LIN {X 0.107,Y -668.681,Z 738.565,A 0.000,B 0.000,C 90.000,E1 317.676} C_DIS
LIN {X 0.186,Y -672.664,Z 738.558,A 0.000,B 0.000,C 90.000,E1 316.458} C_DIS
LIN {X 0.302,Y -676.399,Z 738.552,A 0.000,B 0.000,C 90.000,E1 315.243} C_DIS
LIN {X -0.045,Y -679.125,Z 738.546,A 0.000,B 0.000,C 90.000,E1 314.312} C_DIS
LIN {X 0.190,Y -682.249,Z 738.540,A 0.000,B 0.000,C 90.000,E1 313.095} C_DIS
LIN {X 0.341,Y -684.050,Z 738.536,A 0.000,B 0.000,C 90.000,E1 312.366} C_DIS
LIN {X -0.296,Y -686.830,Z 738.529,A 0.000,B 0.000,C 90.000,E1 311.229} C_DIS
LIN {X 0.079,Y -689.190,Z 738.522,A 0.000,B 0.000,C 90.000,E1 310.011} C_DIS
LIN {X -0.016,Y -690.783,Z 738.517,A 0.000,B 0.000,C 90.000,E1 309.072} C_DIS
LIN {X 0.345,Y -692.184,Z 738.512,A 0.000,B 0.000,C 90.000,E1 308.096} C_DIS
LIN {X 0.292,Y -693.400,Z 738.507,A 0.000,B 0.000,C 90.000,E1 307.156} C_DIS
LIN {X -0.101,Y -694.755,Z 738.500,A 0.000,B 0.000,C 90.000,E1 306.011} C_DIS
LIN {X 0.435,Y -695.668,Z 738.495,A 0.000,B 0.000,C 90.000,E1 305.025} C_DIS
LIN {X -0.332,Y -696.670,Z 738.488,A 0.000,B 0.000,C 90.000,E1 303.913} C_DIS
LIN {X 0.362,Y -697.989,Z 738.479,A 0.000,B 0.000,C 90.000,E1 302.212} C_DIS
LIN {X 0.208,Y -698.942,Z 738.473,A 0.000,B 0.000,C 90.000,E1 301.052} C_DIS
LIN {X 0.041,Y -699.423,Z 738.467,A 0.000,B 0.000,C 90.000,E1 300.129} C_DIS
LIN {X 0.151,Y -699.766,Z 738.461,A 0.000,B 0.000,C 90.000,E1 298.949} C_DIS
LIN {X 0.265,Y -700.096,Z 738.454,A 0.000,B 0.000,C 90.000,E1 297.769} C_DIS
LIN {X 0.057,Y -700.510,Z 738.448,A 0.000,B 0.000,C 90.000,E1 296.616} C_DIS
LIN {X 0.130,Y -701.206,Z 738.440,A 0.000,B 0.000,C 90.000,E1 295.207} C_DIS
LIN {X -0.253,Y -701.147,Z 738.438,A 0.000,B 0.000,C 90.000,E1 294.771} C_DIS
LIN {X 0.020,Y -700.966,Z 738.436,A 0.000,B 0.000,C 90.000,E1 294.515} C_DIS
LIN {X -0.362,Y -700.003,Z 738.434,A 0.000,B 0.000,C 90.000,E1 294.079} C_DIS
LIN {X -0.093,Y -699.108,Z 738.432,A 0.000,B 0.000,C 90.000,E1 293.823} C_DIS
LIN {X -0.107,Y -697.250,Z 738.431,A 0.000,B 0.000,C 90.000,E1 293.590} C_DIS
LIN {X 0.281,Y -694.168,Z 738.429,A 0.000,B 0.000,C 90.000,E1 293.206} C_DIS
LIN {X -0.231,Y -692.628,Z 738.428,A 0.000,B 0.000,C 90.000,E1 293.131} C_DIS
LIN {X -0.206,Y -690.549,Z 738.428,A 0.000,B 0.000,C 90.000,E1 293.025} C_DIS
LIN {X 0.164,Y -686.427,Z 738.427,A 0.000,B 0.000,C 90.000,E1 292.823} C_DIS
LIN {X 0.124,Y -682.661,Z 738.426,A 0.000,B 0.000,C 90.000,E1 292.695} C_DIS
LIN {X -0.149,Y -676.703,Z 738.425,A 0.000,B 0.000,C 90.000,E1 292.567} C_DIS
LIN {X -0.265,Y -668.924,Z 738.425,A 0.000,B 0.000,C 90.000,E1 292.461} C_DIS
LIN {X -0.069,Y -659.282,Z 738.424,A 0.000,B 0.000,C 90.000,E1 292.333} C_DIS
LIN {X -0.387,Y -645.945,Z 738.423,A 0.000,B 0.000,C 90.000,E1 292.153} C_DIS
LIN {X 0.142,Y -632.515,Z 738.421,A 0.000,B 0.000,C 90.000,E1 291.844} C_DIS
LIN {X 0.064,Y -619.307,Z 738.420,A 0.000,B 0.000,C 90.000,E1 291.535} C_DIS
LIN {X 0.213,Y -588.192,Z 738.415,A 0.000,B 0.000,C 90.000,E1 290.663} C_DIS
LIN {X -0.258,Y -574.047,Z 738.413,A 0.000,B 0.000,C 90.000,E1 290.301} C_DIS
LIN {X 0.173,Y -566.696,Z 738.412,A 0.000,B 0.000,C 90.000,E1 290.066} C_DIS
LIN {X 0.081,Y -561.198,Z 738.411,A 0.000,B 0.000,C 90.000,E1 289.885} C_DIS
LIN {X 0.104,Y -556.813,Z 738.409,A 0.000,B 0.000,C 90.000,E1 289.631} C_DIS
LIN {X 0.047,Y -556.755,Z 738.409,A 0.000,B 0.000,C 90.000,E1 289.631} C_DIS
LIN {X 0.005,Y -555.577,Z 738.408,A 0.000,B 0.000,C 90.000,E1 289.450} C_DIS
LIN {X -0.006,Y -554.906,Z 738.406,A 0.000,B 0.000,C 90.000,E1 289.033} C_DIS
LIN {X 0.300,Y -554.456,Z 738.398,A 0.000,B 0.000,C 90.000,E1 287.692} C_DIS
LIN {X 0.241,Y -553.803,Z 738.389,A 0.000,B 0.000,C 90.000,E1 286.024} C_DIS
LIN {X -0.248,Y -553.121,Z 738.378,A 0.000,B 0.000,C 90.000,E1 284.120} C_DIS
LIN {X 0.178,Y -552.515,Z 738.367,A 0.000,B 0.000,C 90.000,E1 282.119} C_DIS
LIN {X 0.126,Y -552.034,Z 738.360,A 0.000,B 0.000,C 90.000,E1 280.725} C_DIS
LIN {X 0.171,Y -551.422,Z 738.352,A 0.000,B 0.000,C 90.000,E1 279.321} C_DIS
LIN {X 0.240,Y -550.474,Z 738.341,A 0.000,B 0.000,C 90.000,E1 277.352} C_DIS
LIN {X 0.211,Y -549.573,Z 738.330,A 0.000,B 0.000,C 90.000,E1 275.391} C_DIS
LIN {X -0.028,Y -548.987,Z 738.322,A 0.000,B 0.000,C 90.000,E1 274.012} C_DIS
LIN {X -0.214,Y -547.965,Z 738.311,A 0.000,B 0.000,C 90.000,E1 272.064} C_DIS
LIN {X -0.008,Y -547.441,Z 738.305,A 0.000,B 0.000,C 90.000,E1 270.917} C_DIS
LIN {X 0.221,Y -546.611,Z 738.297,A 0.000,B 0.000,C 90.000,E1 269.484} C_DIS
LIN {X -0.058,Y -545.522,Z 738.288,A 0.000,B 0.000,C 90.000,E1 267.822} C_DIS
LIN {X 0.248,Y -544.272,Z 738.277,A 0.000,B 0.000,C 90.000,E1 265.812} C_DIS
LIN {X -0.075,Y -543.297,Z 738.269,A 0.000,B 0.000,C 90.000,E1 264.432} C_DIS
LIN {X 0.189,Y -542.025,Z 738.260,A 0.000,B 0.000,C 90.000,E1 262.704} C_DIS
LIN {X -0.126,Y -540.901,Z 738.252,A 0.000,B 0.000,C 90.000,E1 261.319} C_DIS
LIN {X 0.219,Y -539.453,Z 738.242,A 0.000,B 0.000,C 90.000,E1 259.577} C_DIS
LIN {X 0.167,Y -537.839,Z 738.231,A 0.000,B 0.000,C 90.000,E1 257.589} C_DIS
LIN {X 0.076,Y -536.590,Z 738.223,A 0.000,B 0.000,C 90.000,E1 256.172} C_DIS
LIN {X -0.086,Y -535.398,Z 738.217,A 0.000,B 0.000,C 90.000,E1 255.046} C_DIS
LIN {X -0.074,Y -533.864,Z 738.209,A 0.000,B 0.000,C 90.000,E1 253.614} C_DIS
LIN {X -0.092,Y -532.365,Z 738.201,A 0.000,B 0.000,C 90.000,E1 252.181} C_DIS
LIN {X -0.168,Y -531.064,Z 738.195,A 0.000,B 0.000,C 90.000,E1 251.040} C_DIS
LIN {X -0.093,Y -529.518,Z 738.188,A 0.000,B 0.000,C 90.000,E1 249.880} C_DIS
LIN {X 0.141,Y -527.596,Z 738.180,A 0.000,B 0.000,C 90.000,E1 248.411} C_DIS
LIN {X 0.185,Y -526.349,Z 738.175,A 0.000,B 0.000,C 90.000,E1 247.539} C_DIS
LIN {X 0.236,Y -523.743,Z 738.166,A 0.000,B 0.000,C 90.000,E1 245.793} C_DIS
LIN {X -0.029,Y -520.893,Z 738.156,A 0.000,B 0.000,C 90.000,E1 244.076} C_DIS
LIN {X -0.160,Y -518.891,Z 738.150,A 0.000,B 0.000,C 90.000,E1 242.922} C_DIS
LIN {X 0.131,Y -516.673,Z 738.143,A 0.000,B 0.000,C 90.000,E1 241.719} C_DIS
LIN {X 0.080,Y -513.766,Z 738.135,A 0.000,B 0.000,C 90.000,E1 240.255} C_DIS
LIN {X -0.017,Y -510.889,Z 738.127,A 0.000,B 0.000,C 90.000,E1 238.791} C_DIS
LIN {X 0.201,Y -508.495,Z 738.120,A 0.000,B 0.000,C 90.000,E1 237.582} C_DIS
LIN {X -0.049,Y -505.942,Z 738.113,A 0.000,B 0.000,C 90.000,E1 236.421} C_DIS
LIN {X 0.251,Y -502.660,Z 738.105,A 0.000,B 0.000,C 90.000,E1 234.895} C_DIS
LIN {X 0.074,Y -499.029,Z 738.097,A 0.000,B 0.000,C 90.000,E1 233.417} C_DIS
LIN {X 0.126,Y -495.165,Z 738.089,A 0.000,B 0.000,C 90.000,E1 231.904} C_DIS
LIN {X -0.284,Y -491.468,Z 738.080,A 0.000,B 0.000,C 90.000,E1 230.436} C_DIS
LIN {X 0.245,Y -487.936,Z 738.072,A 0.000,B 0.000,C 90.000,E1 228.852} C_DIS
LIN {X -0.125,Y -481.804,Z 738.056,A 0.000,B 0.000,C 90.000,E1 226.134} C_DIS
LIN {X 0.073,Y -477.123,Z 738.044,A 0.000,B 0.000,C 90.000,E1 223.947} C_DIS
LIN {X -0.037,Y -473.885,Z 738.036,A 0.000,B 0.000,C 90.000,E1 222.405} C_DIS
LIN {X 0.107,Y -470.495,Z 738.027,A 0.000,B 0.000,C 90.000,E1 220.825} C_DIS
LIN {X 0.156,Y -464.903,Z 738.013,A 0.000,B 0.000,C 90.000,E1 218.302} C_DIS
LIN {X 0.091,Y -460.160,Z 738.001,A 0.000,B 0.000,C 90.000,E1 216.091} C_DIS
LIN {X -0.258,Y -455.010,Z 737.986,A 0.000,B 0.000,C 90.000,E1 213.579} C_DIS
LIN {X 0.008,Y -452.628,Z 737.979,A 0.000,B 0.000,C 90.000,E1 212.260} C_DIS
LIN {X -0.078,Y -448.964,Z 737.969,A 0.000,B 0.000,C 90.000,E1 210.335} C_DIS
LIN {X 0.144,Y -445.421,Z 737.958,A 0.000,B 0.000,C 90.000,E1 208.359} C_DIS
LIN {X -0.034,Y -442.971,Z 737.950,A 0.000,B 0.000,C 90.000,E1 207.078} C_DIS
LIN {X -0.209,Y -439.876,Z 737.941,A 0.000,B 0.000,C 90.000,E1 205.463} C_DIS
LIN {X -0.005,Y -436.307,Z 737.930,A 0.000,B 0.000,C 90.000,E1 203.462} C_DIS
LIN {X 0.123,Y -433.167,Z 737.921,A 0.000,B 0.000,C 90.000,E1 201.791} C_DIS
LIN {X 0.207,Y -428.839,Z 737.908,A 0.000,B 0.000,C 90.000,E1 199.450} C_DIS
LIN {X 0.082,Y -425.100,Z 737.897,A 0.000,B 0.000,C 90.000,E1 197.457} C_DIS
LIN {X -0.095,Y -422.490,Z 737.890,A 0.000,B 0.000,C 90.000,E1 196.134} C_DIS
LIN {X 0.004,Y -417.440,Z 737.875,A 0.000,B 0.000,C 90.000,E1 193.411} C_DIS
LIN {X -0.006,Y -413.905,Z 737.863,A 0.000,B 0.000,C 90.000,E1 191.366} C_DIS
LIN {X -0.044,Y -409.097,Z 737.848,A 0.000,B 0.000,C 90.000,E1 188.624} C_DIS
LIN {X -0.001,Y -406.349,Z 737.838,A 0.000,B 0.000,C 90.000,E1 186.891} C_DIS
LIN {X -0.200,Y -401.138,Z 737.819,A 0.000,B 0.000,C 90.000,E1 183.440} C_DIS
LIN {X 0.191,Y -397.074,Z 737.801,A 0.000,B 0.000,C 90.000,E1 180.229} C_DIS
LIN {X 0.167,Y -394.437,Z 737.788,A 0.000,B 0.000,C 90.000,E1 177.764} C_DIS
LIN {X 0.080,Y -391.977,Z 737.774,A 0.000,B 0.000,C 90.000,E1 175.298} C_DIS
LIN {X -0.138,Y -389.590,Z 737.756,A 0.000,B 0.000,C 90.000,E1 172.129} C_DIS
LIN {X 0.182,Y -388.175,Z 737.738,A 0.000,B 0.000,C 90.000,E1 168.870} C_DIS
LIN {X -0.080,Y -387.020,Z 737.722,A 0.000,B 0.000,C 90.000,E1 166.047} C_DIS
LIN {X 0.160,Y -386.296,Z 737.709,A 0.000,B 0.000,C 90.000,E1 163.504} C_DIS
LIN {X -0.177,Y -385.941,Z 737.697,A 0.000,B 0.000,C 90.000,E1 161.402} C_DIS
LIN {X 0.070,Y -385.662,Z 737.687,A 0.000,B 0.000,C 90.000,E1 159.571} C_DIS
LIN {X 0.113,Y -385.332,Z 737.675,A 0.000,B 0.000,C 90.000,E1 157.411} C_DIS
LIN {X -0.061,Y -385.252,Z 737.657,A 0.000,B 0.000,C 90.000,E1 154.204} C_DIS
LIN {X -0.062,Y -386.656,Z 737.631,A 0.000,B 0.000,C 90.000,E1 149.537} C_DIS
LIN {X -0.080,Y -389.021,Z 737.611,A 0.000,B 0.000,C 90.000,E1 145.960} C_DIS
LIN {X -0.062,Y -393.045,Z 737.591,A 0.000,B 0.000,C 90.000,E1 142.396} C_DIS
LIN {X 0.038,Y -395.333,Z 737.583,A 0.000,B 0.000,C 90.000,E1 140.964} C_DIS
LIN {X 0.017,Y -397.610,Z 737.577,A 0.000,B 0.000,C 90.000,E1 139.908} C_DIS
LIN {X -0.083,Y -399.603,Z 737.573,A 0.000,B 0.000,C 90.000,E1 139.218} C_DIS
LIN {X 0.085,Y -401.742,Z 737.570,A 0.000,B 0.000,C 90.000,E1 138.609} C_DIS
LIN {X 0.026,Y -405.333,Z 737.566,A 0.000,B 0.000,C 90.000,E1 137.919} C_DIS
LIN {X 0.203,Y -408.142,Z 737.564,A 0.000,B 0.000,C 90.000,E1 137.472} C_DIS
LIN {X -0.041,Y -413.068,Z 737.561,A 0.000,B 0.000,C 90.000,E1 136.905} C_DIS
LIN {X -0.026,Y -430.952,Z 737.550,A 0.000,B 0.000,C 90.000,E1 135.081} C_DIS
LIN {X -0.178,Y -447.096,Z 737.542,A 0.000,B 0.000,C 90.000,E1 133.542} C_DIS
LIN {X 0.034,Y -454.423,Z 737.538,A 0.000,B 0.000,C 90.000,E1 132.813} C_DIS
LIN {X 0.015,Y -465.875,Z 737.532,A 0.000,B 0.000,C 90.000,E1 131.676} C_DIS
LIN {X -0.272,Y -475.659,Z 737.526,A 0.000,B 0.000,C 90.000,E1 130.701} C_DIS
LIN {X 0.068,Y -482.496,Z 737.522,A 0.000,B 0.000,C 90.000,E1 129.930} C_DIS
LIN {X -0.093,Y -487.844,Z 737.519,A 0.000,B 0.000,C 90.000,E1 129.358} C_DIS
LIN {X 0.171,Y -494.069,Z 737.515,A 0.000,B 0.000,C 90.000,E1 128.624} C_DIS
LIN {X 0.041,Y -499.872,Z 737.511,A 0.000,B 0.000,C 90.000,E1 127.935} C_DIS
LIN {X -0.145,Y -503.261,Z 737.508,A 0.000,B 0.000,C 90.000,E1 127.523} C_DIS
LIN {X -0.193,Y -507.501,Z 737.505,A 0.000,B 0.000,C 90.000,E1 126.950} C_DIS
LIN {X 0.241,Y -513.463,Z 737.500,A 0.000,B 0.000,C 90.000,E1 126.011} C_DIS
LIN {X -0.025,Y -516.316,Z 737.498,A 0.000,B 0.000,C 90.000,E1 125.598} C_DIS
LIN {X -0.160,Y -519.847,Z 737.495,A 0.000,B 0.000,C 90.000,E1 125.025} C_DIS
LIN {X -0.014,Y -523.848,Z 737.490,A 0.000,B 0.000,C 90.000,E1 124.278} C_DIS
LIN {X -0.263,Y -527.506,Z 737.486,A 0.000,B 0.000,C 90.000,E1 123.579} C_DIS
LIN {X 0.093,Y -531.525,Z 737.482,A 0.000,B 0.000,C 90.000,E1 122.673} C_DIS
LIN {X 0.070,Y -534.696,Z 737.478,A 0.000,B 0.000,C 90.000,E1 121.957} C_DIS
LIN {X 0.223,Y -539.548,Z 737.471,A 0.000,B 0.000,C 90.000,E1 120.797} C_DIS
LIN {X 0.150,Y -542.982,Z 737.467,A 0.000,B 0.000,C 90.000,E1 119.951} C_DIS
LIN {X -0.118,Y -548.296,Z 737.459,A 0.000,B 0.000,C 90.000,E1 118.565} C_DIS
LIN {X -0.074,Y -552.184,Z 737.452,A 0.000,B 0.000,C 90.000,E1 117.436} C_DIS
LIN {X -0.267,Y -554.861,Z 737.448,A 0.000,B 0.000,C 90.000,E1 116.616} C_DIS
LIN {X 0.317,Y -557.170,Z 737.443,A 0.000,B 0.000,C 90.000,E1 115.720} C_DIS
LIN {X 0.184,Y -559.244,Z 737.438,A 0.000,B 0.000,C 90.000,E1 114.899} C_DIS
LIN {X 0.074,Y -561.035,Z 737.434,A 0.000,B 0.000,C 90.000,E1 114.079} C_DIS
LIN {X 0.295,Y -562.944,Z 737.428,A 0.000,B 0.000,C 90.000,E1 112.950} C_DIS
LIN {X 0.002,Y -564.189,Z 737.423,A 0.000,B 0.000,C 90.000,E1 112.153} C_DIS
LIN {X -0.143,Y -566.243,Z 737.415,A 0.000,B 0.000,C 90.000,E1 110.791} C_DIS
LIN {X 0.079,Y -568.247,Z 737.408,A 0.000,B 0.000,C 90.000,E1 109.396} C_DIS
LIN {X -0.037,Y -570.373,Z 737.399,A 0.000,B 0.000,C 90.000,E1 107.764} C_DIS
LIN {X 0.086,Y -572.007,Z 737.391,A 0.000,B 0.000,C 90.000,E1 106.386} C_DIS
LIN {X 0.233,Y -573.667,Z 737.384,A 0.000,B 0.000,C 90.000,E1 105.009} C_DIS
LIN {X -0.105,Y -575.548,Z 737.375,A 0.000,B 0.000,C 90.000,E1 103.411} C_DIS
LIN {X -0.113,Y -578.115,Z 737.362,A 0.000,B 0.000,C 90.000,E1 101.243} C_DIS
LIN {X -0.040,Y -579.953,Z 737.353,A 0.000,B 0.000,C 90.000,E1 99.613} C_DIS
LIN {X 0.191,Y -581.078,Z 737.347,A 0.000,B 0.000,C 90.000,E1 98.511} C_DIS
LIN {X 0.007,Y -582.404,Z 737.340,A 0.000,B 0.000,C 90.000,E1 97.182} C_DIS
LIN {X 0.010,Y -583.907,Z 737.331,A 0.000,B 0.000,C 90.000,E1 95.568} C_DIS
LIN {X 0.035,Y -585.337,Z 737.322,A 0.000,B 0.000,C 90.000,E1 93.955} C_DIS
LIN {X -0.182,Y -586.393,Z 737.315,A 0.000,B 0.000,C 90.000,E1 92.636} C_DIS
LIN {X 0.014,Y -587.109,Z 737.309,A 0.000,B 0.000,C 90.000,E1 91.547} C_DIS
LIN {X -0.187,Y -587.948,Z 737.301,A 0.000,B 0.000,C 90.000,E1 90.229} C_DIS
LIN {X 0.018,Y -588.478,Z 737.295,A 0.000,B 0.000,C 90.000,E1 89.141} C_DIS
LIN {X 0.055,Y -589.064,Z 737.286,A 0.000,B 0.000,C 90.000,E1 87.535} C_DIS
LIN {X -0.098,Y -589.461,Z 737.279,A 0.000,B 0.000,C 90.000,E1 86.216} C_DIS
LIN {X -0.015,Y -589.727,Z 737.270,A 0.000,B 0.000,C 90.000,E1 84.609} C_DIS
LIN {X 0.123,Y -589.838,Z 737.261,A 0.000,B 0.000,C 90.000,E1 82.996} C_DIS
LIN {X 0.163,Y -589.811,Z 737.254,A 0.000,B 0.000,C 90.000,E1 81.659} C_DIS
LIN {X -0.141,Y -589.707,Z 737.248,A 0.000,B 0.000,C 90.000,E1 80.622} C_DIS
LIN {X 0.327,Y -589.406,Z 737.242,A 0.000,B 0.000,C 90.000,E1 79.511} C_DIS
LIN {X -0.211,Y -588.892,Z 737.235,A 0.000,B 0.000,C 90.000,E1 78.229} C_DIS
LIN {X -0.067,Y -588.264,Z 737.227,A 0.000,B 0.000,C 90.000,E1 76.881} C_DIS
LIN {X 0.203,Y -587.523,Z 737.220,A 0.000,B 0.000,C 90.000,E1 75.519} C_DIS
LIN {X 0.139,Y -586.535,Z 737.211,A 0.000,B 0.000,C 90.000,E1 73.921} C_DIS
LIN {X 0.206,Y -585.339,Z 737.202,A 0.000,B 0.000,C 90.000,E1 72.308} C_DIS
LIN {X 0.207,Y -584.187,Z 737.194,A 0.000,B 0.000,C 90.000,E1 70.967} C_DIS
LIN {X -0.207,Y -583.219,Z 737.188,A 0.000,B 0.000,C 90.000,E1 69.934} C_DIS
LIN {X 0.162,Y -581.544,Z 737.180,A 0.000,B 0.000,C 90.000,E1 68.284} C_DIS
LIN {X -0.083,Y -580.243,Z 737.174,A 0.000,B 0.000,C 90.000,E1 67.230} C_DIS
LIN {X -0.348,Y -578.812,Z 737.167,A 0.000,B 0.000,C 90.000,E1 66.177} C_DIS
LIN {X -0.024,Y -576.791,Z 737.160,A 0.000,B 0.000,C 90.000,E1 64.793} C_DIS
LIN {X -0.106,Y -574.874,Z 737.154,A 0.000,B 0.000,C 90.000,E1 63.717} C_DIS
LIN {X 0.040,Y -572.743,Z 737.148,A 0.000,B 0.000,C 90.000,E1 62.615} C_DIS
LIN {X 0.326,Y -570.910,Z 737.143,A 0.000,B 0.000,C 90.000,E1 61.769} C_DIS
LIN {X -0.080,Y -568.167,Z 737.137,A 0.000,B 0.000,C 90.000,E1 60.717} C_DIS
LIN {X 0.155,Y -565.923,Z 737.133,A 0.000,B 0.000,C 90.000,E1 59.871} C_DIS
LIN {X -0.034,Y -562.551,Z 737.127,A 0.000,B 0.000,C 90.000,E1 58.791} C_DIS
LIN {X 0.126,Y -559.818,Z 737.122,A 0.000,B 0.000,C 90.000,E1 57.946} C_DIS
LIN {X -0.005,Y -557.906,Z 737.119,A 0.000,B 0.000,C 90.000,E1 57.406} C_DIS
LIN {X -0.077,Y -554.656,Z 737.114,A 0.000,B 0.000,C 90.000,E1 56.580} C_DIS
LIN {X 0.131,Y -550.989,Z 737.110,A 0.000,B 0.000,C 90.000,E1 55.722} C_DIS
LIN {X 0.117,Y -547.655,Z 737.106,A 0.000,B 0.000,C 90.000,E1 55.022} C_DIS
LIN {X -0.105,Y -544.774,Z 737.103,A 0.000,B 0.000,C 90.000,E1 54.482} C_DIS
LIN {X -0.175,Y -540.842,Z 737.099,A 0.000,B 0.000,C 90.000,E1 53.783} C_DIS
LIN {X -0.132,Y -537.510,Z 737.096,A 0.000,B 0.000,C 90.000,E1 53.210} C_DIS
LIN {X -0.111,Y -533.843,Z 737.092,A 0.000,B 0.000,C 90.000,E1 52.637} C_DIS
LIN {X -0.118,Y -529.738,Z 737.089,A 0.000,B 0.000,C 90.000,E1 52.065} C_DIS
LIN {X 0.170,Y -525.193,Z 737.086,A 0.000,B 0.000,C 90.000,E1 51.457} C_DIS
LIN {X 0.060,Y -520.379,Z 737.083,A 0.000,B 0.000,C 90.000,E1 50.928} C_DIS
LIN {X 0.044,Y -516.397,Z 737.081,A 0.000,B 0.000,C 90.000,E1 50.517} C_DIS
LIN {X 0.111,Y -509.819,Z 737.077,A 0.000,B 0.000,C 90.000,E1 49.908} C_DIS
LIN {X -0.066,Y -505.289,Z 737.075,A 0.000,B 0.000,C 90.000,E1 49.542} C_DIS
LIN {X 0.035,Y -499.061,Z 737.073,A 0.000,B 0.000,C 90.000,E1 49.057} C_DIS
LIN {X 0.053,Y -491.005,Z 737.069,A 0.000,B 0.000,C 90.000,E1 48.485} C_DIS
LIN {X -0.141,Y -484.512,Z 737.067,A 0.000,B 0.000,C 90.000,E1 48.081} C_DIS
LIN {X 0.101,Y -471.388,Z 737.063,A 0.000,B 0.000,C 90.000,E1 47.229} C_DIS
LIN {X -0.020,Y -448.714,Z 737.055,A 0.000,B 0.000,C 90.000,E1 45.810} C_DIS
LIN {X 0.112,Y -422.909,Z 737.045,A 0.000,B 0.000,C 90.000,E1 44.028} C_DIS
LIN {X 0.094,Y -415.340,Z 737.041,A 0.000,B 0.000,C 90.000,E1 43.419} C_DIS
LIN {X 0.066,Y -415.330,Z 737.041,A 0.000,B 0.000,C 90.000,E1 43.419} C_DIS
LIN {X -0.049,Y -406.477,Z 737.016,A 0.000,B 0.000,C 90.000,E1 38.874} C_DIS
LIN {X -0.158,Y -405.926,Z 737.014,A 0.000,B 0.000,C 90.000,E1 38.543} C_DIS
LIN {X -0.031,Y -403.512,Z 737.008,A 0.000,B 0.000,C 90.000,E1 37.397} C_DIS
LIN {X 0.140,Y -403.957,Z 736.991,A 0.000,B 0.000,C 90.000,E1 34.326} C_DIS
LIN {X -0.121,Y -404.821,Z 736.977,A 0.000,B 0.000,C 90.000,E1 31.926} C_DIS
LIN {X 0.210,Y -405.813,Z 736.966,A 0.000,B 0.000,C 90.000,E1 29.795} C_DIS
LIN {X 0.079,Y -407.078,Z 736.952,A 0.000,B 0.000,C 90.000,E1 27.385} C_DIS
LIN {X 0.158,Y -408.606,Z 736.939,A 0.000,B 0.000,C 90.000,E1 24.951} C_DIS
LIN {X 0.030,Y -410.239,Z 736.927,A 0.000,B 0.000,C 90.000,E1 22.898} C_DIS
LIN {X 0.072,Y -412.511,Z 736.914,A 0.000,B 0.000,C 90.000,E1 20.482} C_DIS
LIN {X 0.046,Y -416.022,Z 736.897,A 0.000,B 0.000,C 90.000,E1 17.402} C_DIS
LIN {X -0.063,Y -418.709,Z 736.885,A 0.000,B 0.000,C 90.000,E1 15.371} C_DIS
LIN {X 0.188,Y -421.626,Z 736.874,A 0.000,B 0.000,C 90.000,E1 13.300} C_DIS
LIN {X -0.007,Y -424.693,Z 736.863,A 0.000,B 0.000,C 90.000,E1 11.299} C_DIS
LIN {X 0.119,Y -427.793,Z 736.852,A 0.000,B 0.000,C 90.000,E1 9.265} C_DIS
LIN {X -0.170,Y -430.896,Z 736.840,A 0.000,B 0.000,C 90.000,E1 7.296} C_DIS
LIN {X 0.064,Y -434.575,Z 736.828,A 0.000,B 0.000,C 90.000,E1 4.935} C_DIS
LIN {X -0.069,Y -438.500,Z 736.815,A 0.000,B 0.000,C 90.000,E1 2.636} C_DIS
LIN {X 0.182,Y -442.154,Z 736.804,A 0.000,B 0.000,C 90.000,E1 0.630} C_DIS
LIN {X -0.037,Y -446.965,Z 736.790,A 0.000,B 0.000,C 90.000,E1 358.165} C_DIS
LIN {X -0.138,Y -452.296,Z 736.775,A 0.000,B 0.000,C 90.000,E1 355.584} C_DIS
LIN {X 0.052,Y -456.611,Z 736.765,A 0.000,B 0.000,C 90.000,E1 353.628} C_DIS
LIN {X -0.069,Y -460.780,Z 736.754,A 0.000,B 0.000,C 90.000,E1 351.724} C_DIS
LIN {X -0.005,Y -463.489,Z 736.747,A 0.000,B 0.000,C 90.000,E1 350.443} C_DIS
LIN {X -0.088,Y -466.597,Z 736.738,A 0.000,B 0.000,C 90.000,E1 348.870} C_DIS
LIN {X -0.204,Y -468.386,Z 736.733,A 0.000,B 0.000,C 90.000,E1 347.937} C_DIS
LIN {X -0.171,Y -471.837,Z 736.722,A 0.000,B 0.000,C 90.000,E1 346.047} C_DIS
LIN {X -0.011,Y -477.883,Z 736.705,A 0.000,B 0.000,C 90.000,E1 342.906} C_DIS
LIN {X -0.222,Y -480.307,Z 736.700,A 0.000,B 0.000,C 90.000,E1 342.000} C_DIS
LIN {X -0.013,Y -481.870,Z 736.697,A 0.000,B 0.000,C 90.000,E1 341.511} C_DIS
LIN {X 0.222,Y -483.602,Z 736.695,A 0.000,B 0.000,C 90.000,E1 341.094} C_DIS
LIN {X -0.163,Y -486.167,Z 736.693,A 0.000,B 0.000,C 90.000,E1 340.678} C_DIS
LIN {X -0.214,Y -489.783,Z 736.690,A 0.000,B 0.000,C 90.000,E1 340.188} C_DIS
LIN {X 0.191,Y -494.013,Z 736.687,A 0.000,B 0.000,C 90.000,E1 339.699} C_DIS
LIN {X 0.161,Y -499.202,Z 736.685,A 0.000,B 0.000,C 90.000,E1 339.263} C_DIS
LIN {X 0.011,Y -508.267,Z 736.681,A 0.000,B 0.000,C 90.000,E1 338.646} C_DIS
LIN {X 0.052,Y -537.192,Z 736.672,A 0.000,B 0.000,C 90.000,E1 336.869} C_DIS
LIN {X -0.132,Y -543.313,Z 736.669,A 0.000,B 0.000,C 90.000,E1 336.485} C_DIS
LIN {X -0.009,Y -550.370,Z 736.666,A 0.000,B 0.000,C 90.000,E1 335.921} C_DIS
LIN {X 0.117,Y -555.868,Z 736.664,A 0.000,B 0.000,C 90.000,E1 335.433} C_DIS
LIN {X 0.191,Y -561.163,Z 736.661,A 0.000,B 0.000,C 90.000,E1 334.921} C_DIS
LIN {X 0.130,Y -566.354,Z 736.658,A 0.000,B 0.000,C 90.000,E1 334.409} C_DIS
LIN {X -0.119,Y -572.539,Z 736.654,A 0.000,B 0.000,C 90.000,E1 333.768} C_DIS
LIN {X 0.093,Y -578.521,Z 736.651,A 0.000,B 0.000,C 90.000,E1 333.076} C_DIS
LIN {X 0.004,Y -584.257,Z 736.647,A 0.000,B 0.000,C 90.000,E1 332.410} C_DIS
LIN {X 0.103,Y -591.843,Z 736.642,A 0.000,B 0.000,C 90.000,E1 331.463} C_DIS
LIN {X 0.047,Y -598.958,Z 736.636,A 0.000,B 0.000,C 90.000,E1 330.539} C_DIS
LIN {X 0.046,Y -606.783,Z 736.631,A 0.000,B 0.000,C 90.000,E1 329.488} C_DIS
LIN {X -0.037,Y -613.185,Z 736.625,A 0.000,B 0.000,C 90.000,E1 328.584} C_DIS
LIN {X 0.164,Y -619.229,Z 736.620,A 0.000,B 0.000,C 90.000,E1 327.661} C_DIS
LIN {X -0.096,Y -624.940,Z 736.615,A 0.000,B 0.000,C 90.000,E1 326.786} C_DIS
LIN {X 0.049,Y -630.251,Z 736.611,A 0.000,B 0.000,C 90.000,E1 325.881} C_DIS
LIN {X -0.106,Y -633.941,Z 736.607,A 0.000,B 0.000,C 90.000,E1 325.261} C_DIS
LIN {X -0.362,Y -639.409,Z 736.601,A 0.000,B 0.000,C 90.000,E1 324.276} C_DIS
LIN {X -0.164,Y -644.604,Z 736.596,A 0.000,B 0.000,C 90.000,E1 323.256} C_DIS
LIN {X 0.196,Y -648.259,Z 736.592,A 0.000,B 0.000,C 90.000,E1 322.477} C_DIS
LIN {X 0.026,Y -653.425,Z 736.586,A 0.000,B 0.000,C 90.000,E1 321.376} C_DIS
LIN {X -0.047,Y -656.652,Z 736.581,A 0.000,B 0.000,C 90.000,E1 320.642} C_DIS
LIN {X 0.349,Y -661.743,Z 736.575,A 0.000,B 0.000,C 90.000,E1 319.380} C_DIS
LIN {X -0.163,Y -665.584,Z 736.569,A 0.000,B 0.000,C 90.000,E1 318.447} C_DIS
LIN {X -0.132,Y -668.241,Z 736.565,A 0.000,B 0.000,C 90.000,E1 317.715} C_DIS
LIN {X -0.096,Y -672.263,Z 736.558,A 0.000,B 0.000,C 90.000,E1 316.500} C_DIS
LIN {X 0.026,Y -676.034,Z 736.552,A 0.000,B 0.000,C 90.000,E1 315.283} C_DIS
LIN {X -0.323,Y -678.836,Z 736.546,A 0.000,B 0.000,C 90.000,E1 314.352} C_DIS
LIN {X -0.160,Y -681.400,Z 736.541,A 0.000,B 0.000,C 90.000,E1 313.380} C_DIS
LIN {X 0.071,Y -683.851,Z 736.536,A 0.000,B 0.000,C 90.000,E1 312.405} C_DIS
LIN {X -0.108,Y -686.684,Z 736.529,A 0.000,B 0.000,C 90.000,E1 311.229} C_DIS
LIN {X 0.266,Y -689.113,Z 736.522,A 0.000,B 0.000,C 90.000,E1 310.011} C_DIS
LIN {X 0.170,Y -690.761,Z 736.517,A 0.000,B 0.000,C 90.000,E1 309.072} C_DIS
LIN {X -0.012,Y -692.200,Z 736.512,A 0.000,B 0.000,C 90.000,E1 308.141} C_DIS
LIN {X -0.071,Y -693.442,Z 736.507,A 0.000,B 0.000,C 90.000,E1 307.202} C_DIS
LIN {X 0.088,Y -694.834,Z 736.500,A 0.000,B 0.000,C 90.000,E1 306.011} C_DIS
LIN {X -0.344,Y -695.752,Z 736.495,A 0.000,B 0.000,C 90.000,E1 305.105} C_DIS
LIN {X 0.206,Y -696.584,Z 736.490,A 0.000,B 0.000,C 90.000,E1 304.119} C_DIS
LIN {X -0.034,Y -698.105,Z 736.479,A 0.000,B 0.000,C 90.000,E1 302.260} C_DIS
LIN {X 0.044,Y -699.056,Z 736.473,A 0.000,B 0.000,C 90.000,E1 301.082} C_DIS
LIN {X 0.240,Y -699.549,Z 736.468,A 0.000,B 0.000,C 90.000,E1 300.129} C_DIS
LIN {X 0.084,Y -699.851,Z 736.462,A 0.000,B 0.000,C 90.000,E1 299.205} C_DIS
LIN {X -0.151,Y -700.202,Z 736.455,A 0.000,B 0.000,C 90.000,E1 297.820} C_DIS
LIN {X -0.129,Y -700.835,Z 736.445,A 0.000,B 0.000,C 90.000,E1 296.181} C_DIS
LIN {X 0.337,Y -701.314,Z 736.440,A 0.000,B 0.000,C 90.000,E1 295.207} C_DIS
LIN {X -0.045,Y -701.262,Z 736.438,A 0.000,B 0.000,C 90.000,E1 294.771} C_DIS
LIN {X 0.229,Y -701.124,Z 736.436,A 0.000,B 0.000,C 90.000,E1 294.515} C_DIS
LIN {X -0.153,Y -700.068,Z 736.434,A 0.000,B 0.000,C 90.000,E1 294.079} C_DIS
LIN {X 0.116,Y -699.208,Z 736.432,A 0.000,B 0.000,C 90.000,E1 293.823} C_DIS
LIN {X 0.249,Y -698.389,Z 736.432,A 0.000,B 0.000,C 90.000,E1 293.695} C_DIS
LIN {X -0.276,Y -695.325,Z 736.430,A 0.000,B 0.000,C 90.000,E1 293.387} C_DIS
LIN {X -0.149,Y -694.162,Z 736.429,A 0.000,B 0.000,C 90.000,E1 293.259} C_DIS
LIN {X -0.023,Y -692.692,Z 736.429,A 0.000,B 0.000,C 90.000,E1 293.131} C_DIS
LIN {X -0.029,Y -690.550,Z 736.428,A 0.000,B 0.000,C 90.000,E1 293.025} C_DIS
LIN {X 0.314,Y -686.326,Z 736.427,A 0.000,B 0.000,C 90.000,E1 292.823} C_DIS
LIN {X 0.063,Y -682.540,Z 736.426,A 0.000,B 0.000,C 90.000,E1 292.717} C_DIS
LIN {X -0.189,Y -676.686,Z 736.425,A 0.000,B 0.000,C 90.000,E1 292.589} C_DIS
LIN {X -0.039,Y -668.795,Z 736.425,A 0.000,B 0.000,C 90.000,E1 292.461} C_DIS
LIN {X 0.032,Y -662.324,Z 736.424,A 0.000,B 0.000,C 90.000,E1 292.386} C_DIS
LIN {X -0.107,Y -649.370,Z 736.423,A 0.000,B 0.000,C 90.000,E1 292.206} C_DIS
LIN {X -0.034,Y -635.909,Z 736.422,A 0.000,B 0.000,C 90.000,E1 291.950} C_DIS
LIN {X 0.113,Y -626.022,Z 736.421,A 0.000,B 0.000,C 90.000,E1 291.716} C_DIS
LIN {X -0.021,Y -602.027,Z 736.417,A 0.000,B 0.000,C 90.000,E1 291.099} C_DIS
LIN {X 0.164,Y -577.468,Z 736.413,A 0.000,B 0.000,C 90.000,E1 290.375} C_DIS
LIN {X 0.147,Y -569.910,Z 736.412,A 0.000,B 0.000,C 90.000,E1 290.174} C_DIS
LIN {X -0.212,Y -566.653,Z 736.412,A 0.000,B 0.000,C 90.000,E1 290.120} C_DIS
LIN {X 0.215,Y -561.107,Z 736.411,A 0.000,B 0.000,C 90.000,E1 289.885} C_DIS
LIN {X 0.211,Y -556.729,Z 736.409,A 0.000,B 0.000,C 90.000,E1 289.631} C_DIS
LIN {X 0.154,Y -556.667,Z 736.409,A 0.000,B 0.000,C 90.000,E1 289.631} C_DIS
LIN {X -0.051,Y -555.554,Z 736.408,A 0.000,B 0.000,C 90.000,E1 289.450} C_DIS
LIN {X -0.063,Y -554.904,Z 736.406,A 0.000,B 0.000,C 90.000,E1 289.033} C_DIS
LIN {X 0.073,Y -554.450,Z 736.399,A 0.000,B 0.000,C 90.000,E1 287.764} C_DIS
LIN {X 0.178,Y -553.821,Z 736.389,A 0.000,B 0.000,C 90.000,E1 286.079} C_DIS
LIN {X 0.221,Y -553.106,Z 736.379,A 0.000,B 0.000,C 90.000,E1 284.120} C_DIS
LIN {X -0.132,Y -552.580,Z 736.369,A 0.000,B 0.000,C 90.000,E1 282.479} C_DIS
LIN {X -0.068,Y -552.118,Z 736.362,A 0.000,B 0.000,C 90.000,E1 281.074} C_DIS
LIN {X -0.021,Y -551.540,Z 736.354,A 0.000,B 0.000,C 90.000,E1 279.670} C_DIS
LIN {X -0.087,Y -550.841,Z 736.346,A 0.000,B 0.000,C 90.000,E1 278.276} C_DIS
LIN {X -0.246,Y -550.208,Z 736.338,A 0.000,B 0.000,C 90.000,E1 276.891} C_DIS
LIN {X 0.216,Y -549.356,Z 736.327,A 0.000,B 0.000,C 90.000,E1 274.878} C_DIS
LIN {X -0.149,Y -549.012,Z 736.323,A 0.000,B 0.000,C 90.000,E1 274.073} C_DIS
LIN {X 0.250,Y -548.021,Z 736.312,A 0.000,B 0.000,C 90.000,E1 272.064} C_DIS
LIN {X -0.090,Y -547.503,Z 736.305,A 0.000,B 0.000,C 90.000,E1 270.974} C_DIS
LIN {X 0.140,Y -546.681,Z 736.298,A 0.000,B 0.000,C 90.000,E1 269.542} C_DIS
LIN {X -0.137,Y -545.609,Z 736.288,A 0.000,B 0.000,C 90.000,E1 267.879} C_DIS
LIN {X 0.172,Y -544.341,Z 736.277,A 0.000,B 0.000,C 90.000,E1 265.869} C_DIS
LIN {X -0.148,Y -543.375,Z 736.269,A 0.000,B 0.000,C 90.000,E1 264.489} C_DIS
LIN {X 0.119,Y -542.115,Z 736.260,A 0.000,B 0.000,C 90.000,E1 262.761} C_DIS
LIN {X -0.191,Y -540.959,Z 736.252,A 0.000,B 0.000,C 90.000,E1 261.376} C_DIS
LIN {X 0.158,Y -539.528,Z 736.243,A 0.000,B 0.000,C 90.000,E1 259.634} C_DIS
LIN {X 0.175,Y -537.693,Z 736.230,A 0.000,B 0.000,C 90.000,E1 257.353} C_DIS
LIN {X 0.084,Y -536.416,Z 736.222,A 0.000,B 0.000,C 90.000,E1 255.936} C_DIS
LIN {X 0.159,Y -534.581,Z 736.212,A 0.000,B 0.000,C 90.000,E1 254.212} C_DIS
LIN {X -0.128,Y -532.449,Z 736.201,A 0.000,B 0.000,C 90.000,E1 252.236} C_DIS
LIN {X -0.201,Y -531.179,Z 736.195,A 0.000,B 0.000,C 90.000,E1 251.094} C_DIS
LIN {X -0.120,Y -529.646,Z 736.188,A 0.000,B 0.000,C 90.000,E1 249.934} C_DIS
LIN {X 0.122,Y -527.721,Z 736.180,A 0.000,B 0.000,C 90.000,E1 248.465} C_DIS
LIN {X -0.031,Y -526.478,Z 736.176,A 0.000,B 0.000,C 90.000,E1 247.614} C_DIS
LIN {X -0.148,Y -524.299,Z 736.168,A 0.000,B 0.000,C 90.000,E1 246.177} C_DIS
LIN {X 0.077,Y -522.934,Z 736.163,A 0.000,B 0.000,C 90.000,E1 245.281} C_DIS
LIN {X -0.107,Y -520.551,Z 736.155,A 0.000,B 0.000,C 90.000,E1 243.845} C_DIS
LIN {X 0.076,Y -519.041,Z 736.150,A 0.000,B 0.000,C 90.000,E1 242.948} C_DIS
LIN {X 0.150,Y -516.806,Z 736.143,A 0.000,B 0.000,C 90.000,E1 241.769} C_DIS
LIN {X -0.149,Y -513.907,Z 736.135,A 0.000,B 0.000,C 90.000,E1 240.333} C_DIS
LIN {X -0.246,Y -511.023,Z 736.127,A 0.000,B 0.000,C 90.000,E1 238.869} C_DIS
LIN {X -0.030,Y -508.611,Z 736.120,A 0.000,B 0.000,C 90.000,E1 237.661} C_DIS
LIN {X 0.038,Y -505.437,Z 736.112,A 0.000,B 0.000,C 90.000,E1 236.167} C_DIS
LIN {X 0.022,Y -502.806,Z 736.105,A 0.000,B 0.000,C 90.000,E1 234.975} C_DIS
LIN {X -0.153,Y -499.199,Z 736.097,A 0.000,B 0.000,C 90.000,E1 233.497} C_DIS
LIN {X -0.100,Y -495.350,Z 736.089,A 0.000,B 0.000,C 90.000,E1 231.984} C_DIS
LIN {X 0.187,Y -491.635,Z 736.080,A 0.000,B 0.000,C 90.000,E1 230.436} C_DIS
LIN {X 0.178,Y -487.356,Z 736.070,A 0.000,B 0.000,C 90.000,E1 228.609} C_DIS
LIN {X -0.003,Y -481.925,Z 736.057,A 0.000,B 0.000,C 90.000,E1 226.176} C_DIS
LIN {X -0.135,Y -477.246,Z 736.045,A 0.000,B 0.000,C 90.000,E1 224.028} C_DIS
LIN {X 0.080,Y -473.975,Z 736.036,A 0.000,B 0.000,C 90.000,E1 222.447} C_DIS
LIN {X -0.177,Y -471.299,Z 736.029,A 0.000,B 0.000,C 90.000,E1 221.229} C_DIS
LIN {X 0.022,Y -467.080,Z 736.018,A 0.000,B 0.000,C 90.000,E1 219.322} C_DIS
LIN {X 0.135,Y -463.659,Z 736.010,A 0.000,B 0.000,C 90.000,E1 217.729} C_DIS
LIN {X 0.039,Y -458.943,Z 735.997,A 0.000,B 0.000,C 90.000,E1 215.518} C_DIS
LIN {X 0.127,Y -453.341,Z 735.981,A 0.000,B 0.000,C 90.000,E1 212.625} C_DIS
LIN {X -0.008,Y -449.121,Z 735.969,A 0.000,B 0.000,C 90.000,E1 210.384} C_DIS
LIN {X 0.063,Y -444.949,Z 735.956,A 0.000,B 0.000,C 90.000,E1 208.103} C_DIS
LIN {X -0.031,Y -441.276,Z 735.945,A 0.000,B 0.000,C 90.000,E1 206.155} C_DIS
LIN {X 0.214,Y -437.029,Z 735.933,A 0.000,B 0.000,C 90.000,E1 203.823} C_DIS
LIN {X -0.053,Y -433.928,Z 735.923,A 0.000,B 0.000,C 90.000,E1 202.206} C_DIS
LIN {X 0.086,Y -430.188,Z 735.912,A 0.000,B 0.000,C 90.000,E1 200.194} C_DIS
LIN {X 0.134,Y -427.738,Z 735.905,A 0.000,B 0.000,C 90.000,E1 198.852} C_DIS
LIN {X 0.132,Y -425.262,Z 735.897,A 0.000,B 0.000,C 90.000,E1 197.511} C_DIS
LIN {X -0.164,Y -422.659,Z 735.890,A 0.000,B 0.000,C 90.000,E1 196.205} C_DIS
LIN {X -0.044,Y -417.622,Z 735.875,A 0.000,B 0.000,C 90.000,E1 193.480} C_DIS
LIN {X -0.004,Y -414.674,Z 735.865,A 0.000,B 0.000,C 90.000,E1 191.771} C_DIS
LIN {X -0.020,Y -409.864,Z 735.850,A 0.000,B 0.000,C 90.000,E1 189.029} C_DIS
LIN {X 0.052,Y -406.521,Z 735.839,A 0.000,B 0.000,C 90.000,E1 186.947} C_DIS
LIN {X -0.088,Y -402.291,Z 735.823,A 0.000,B 0.000,C 90.000,E1 184.188} C_DIS
LIN {X 0.014,Y -398.501,Z 735.808,A 0.000,B 0.000,C 90.000,E1 181.375} C_DIS
LIN {X -0.044,Y -395.349,Z 735.792,A 0.000,B 0.000,C 90.000,E1 178.568} C_DIS
LIN {X -0.030,Y -393.183,Z 735.780,A 0.000,B 0.000,C 90.000,E1 176.445} C_DIS
LIN {X -0.001,Y -390.046,Z 735.759,A 0.000,B 0.000,C 90.000,E1 172.534} C_DIS
LIN {X -0.180,Y -388.356,Z 735.739,A 0.000,B 0.000,C 90.000,E1 168.993} C_DIS
LIN {X 0.000,Y -387.347,Z 735.725,A 0.000,B 0.000,C 90.000,E1 166.464} C_DIS
LIN {X -0.069,Y -386.794,Z 735.715,A 0.000,B 0.000,C 90.000,E1 164.685} C_DIS
LIN {X -0.105,Y -386.300,Z 735.701,A 0.000,B 0.000,C 90.000,E1 162.181} C_DIS
LIN {X 0.023,Y -386.028,Z 735.691,A 0.000,B 0.000,C 90.000,E1 160.369} C_DIS
LIN {X 0.091,Y -385.641,Z 735.677,A 0.000,B 0.000,C 90.000,E1 157.847} C_DIS
LIN {X -0.060,Y -385.471,Z 735.663,A 0.000,B 0.000,C 90.000,E1 155.357} C_DIS
LIN {X 0.095,Y -386.109,Z 735.641,A 0.000,B 0.000,C 90.000,E1 151.385} C_DIS
LIN {X 0.137,Y -387.133,Z 735.627,A 0.000,B 0.000,C 90.000,E1 148.869} C_DIS
LIN {X 0.133,Y -389.091,Z 735.611,A 0.000,B 0.000,C 90.000,E1 146.008} C_DIS
LIN {X 0.006,Y -392.089,Z 735.595,A 0.000,B 0.000,C 90.000,E1 143.176} C_DIS
LIN {X 0.011,Y -393.550,Z 735.590,A 0.000,B 0.000,C 90.000,E1 142.110} C_DIS
LIN {X -0.188,Y -395.813,Z 735.582,A 0.000,B 0.000,C 90.000,E1 140.723} C_DIS
LIN {X 0.001,Y -397.276,Z 735.578,A 0.000,B 0.000,C 90.000,E1 139.989} C_DIS
LIN {X 0.104,Y -399.557,Z 735.573,A 0.000,B 0.000,C 90.000,E1 139.094} C_DIS
LIN {X 0.022,Y -402.113,Z 735.569,A 0.000,B 0.000,C 90.000,E1 138.405} C_DIS
LIN {X 0.049,Y -404.695,Z 735.566,A 0.000,B 0.000,C 90.000,E1 137.877} C_DIS
LIN {X -0.097,Y -407.412,Z 735.564,A 0.000,B 0.000,C 90.000,E1 137.472} C_DIS
LIN {X 0.068,Y -411.994,Z 735.560,A 0.000,B 0.000,C 90.000,E1 136.863} C_DIS
LIN {X 0.134,Y -419.431,Z 735.556,A 0.000,B 0.000,C 90.000,E1 136.053} C_DIS
LIN {X -0.055,Y -432.380,Z 735.549,A 0.000,B 0.000,C 90.000,E1 134.798} C_DIS
LIN {X -0.062,Y -447.159,Z 735.541,A 0.000,B 0.000,C 90.000,E1 133.380} C_DIS
LIN {X -0.247,Y -452.975,Z 735.538,A 0.000,B 0.000,C 90.000,E1 132.852} C_DIS
LIN {X -0.173,Y -458.653,Z 735.535,A 0.000,B 0.000,C 90.000,E1 132.285} C_DIS
LIN {X -0.157,Y -467.203,Z 735.530,A 0.000,B 0.000,C 90.000,E1 131.434} C_DIS
LIN {X -0.026,Y -476.972,Z 735.525,A 0.000,B 0.000,C 90.000,E1 130.415} C_DIS
LIN {X -0.123,Y -482.456,Z 735.521,A 0.000,B 0.000,C 90.000,E1 129.850} C_DIS
LIN {X 0.017,Y -490.509,Z 735.516,A 0.000,B 0.000,C 90.000,E1 128.955} C_DIS
LIN {X -0.180,Y -495.690,Z 735.513,A 0.000,B 0.000,C 90.000,E1 128.382} C_DIS
LIN {X 0.161,Y -499.479,Z 735.511,A 0.000,B 0.000,C 90.000,E1 127.890} C_DIS
LIN {X -0.064,Y -504.127,Z 735.507,A 0.000,B 0.000,C 90.000,E1 127.317} C_DIS
LIN {X -0.061,Y -507.434,Z 735.505,A 0.000,B 0.000,C 90.000,E1 126.870} C_DIS
LIN {X -0.090,Y -512.462,Z 735.501,A 0.000,B 0.000,C 90.000,E1 126.137} C_DIS
LIN {X 0.165,Y -516.310,Z 735.497,A 0.000,B 0.000,C 90.000,E1 125.518} C_DIS
LIN {X 0.030,Y -519.832,Z 735.494,A 0.000,B 0.000,C 90.000,E1 124.945} C_DIS
LIN {X -0.090,Y -523.800,Z 735.490,A 0.000,B 0.000,C 90.000,E1 124.246} C_DIS
LIN {X 0.096,Y -527.483,Z 735.486,A 0.000,B 0.000,C 90.000,E1 123.499} C_DIS
LIN {X -0.128,Y -530.918,Z 735.482,A 0.000,B 0.000,C 90.000,E1 122.801} C_DIS
LIN {X -0.158,Y -534.144,Z 735.478,A 0.000,B 0.000,C 90.000,E1 122.084} C_DIS
LIN {X -0.158,Y -539.609,Z 735.471,A 0.000,B 0.000,C 90.000,E1 120.797} C_DIS
LIN {X 0.038,Y -543.027,Z 735.466,A 0.000,B 0.000,C 90.000,E1 119.922} C_DIS
LIN {X -0.254,Y -547.333,Z 735.460,A 0.000,B 0.000,C 90.000,E1 118.821} C_DIS
LIN {X 0.264,Y -551.383,Z 735.454,A 0.000,B 0.000,C 90.000,E1 117.641} C_DIS
LIN {X 0.090,Y -555.014,Z 735.448,A 0.000,B 0.000,C 90.000,E1 116.539} C_DIS
LIN {X -0.069,Y -557.349,Z 735.443,A 0.000,B 0.000,C 90.000,E1 115.720} C_DIS
LIN {X -0.201,Y -559.418,Z 735.438,A 0.000,B 0.000,C 90.000,E1 114.899} C_DIS
LIN {X 0.201,Y -561.226,Z 735.434,A 0.000,B 0.000,C 90.000,E1 114.027} C_DIS
LIN {X 0.111,Y -562.734,Z 735.429,A 0.000,B 0.000,C 90.000,E1 113.206} C_DIS
LIN {X 0.142,Y -564.422,Z 735.423,A 0.000,B 0.000,C 90.000,E1 112.099} C_DIS
LIN {X -0.190,Y -566.910,Z 735.414,A 0.000,B 0.000,C 90.000,E1 110.482} C_DIS
LIN {X -0.298,Y -568.531,Z 735.408,A 0.000,B 0.000,C 90.000,E1 109.396} C_DIS
LIN {X 0.309,Y -570.707,Z 735.398,A 0.000,B 0.000,C 90.000,E1 107.692} C_DIS
LIN {X 0.064,Y -572.660,Z 735.389,A 0.000,B 0.000,C 90.000,E1 106.079} C_DIS
LIN {X 0.067,Y -574.319,Z 735.382,A 0.000,B 0.000,C 90.000,E1 104.717} C_DIS
LIN {X 0.100,Y -575.920,Z 735.374,A 0.000,B 0.000,C 90.000,E1 103.355} C_DIS
LIN {X -0.108,Y -578.171,Z 735.364,A 0.000,B 0.000,C 90.000,E1 101.478} C_DIS
LIN {X -0.030,Y -580.117,Z 735.355,A 0.000,B 0.000,C 90.000,E1 99.849} C_DIS
LIN {X -0.142,Y -581.545,Z 735.347,A 0.000,B 0.000,C 90.000,E1 98.511} C_DIS
LIN {X -0.091,Y -583.125,Z 735.338,A 0.000,B 0.000,C 90.000,E1 96.891} C_DIS
LIN {X -0.306,Y -584.388,Z 735.331,A 0.000,B 0.000,C 90.000,E1 95.568} C_DIS
LIN {X -0.272,Y -585.832,Z 735.322,A 0.000,B 0.000,C 90.000,E1 93.955} C_DIS
LIN {X -0.084,Y -586.702,Z 735.316,A 0.000,B 0.000,C 90.000,E1 92.865} C_DIS
LIN {X 0.114,Y -587.495,Z 735.310,A 0.000,B 0.000,C 90.000,E1 91.776} C_DIS
LIN {X 0.118,Y -588.486,Z 735.301,A 0.000,B 0.000,C 90.000,E1 90.172} C_DIS
LIN {X -0.058,Y -589.141,Z 735.294,A 0.000,B 0.000,C 90.000,E1 88.854} C_DIS
LIN {X 0.190,Y -589.801,Z 735.283,A 0.000,B 0.000,C 90.000,E1 86.963} C_DIS
LIN {X 0.084,Y -590.065,Z 735.276,A 0.000,B 0.000,C 90.000,E1 85.641} C_DIS
LIN {X -0.261,Y -590.240,Z 735.270,A 0.000,B 0.000,C 90.000,E1 84.609} C_DIS
LIN {X -0.112,Y -590.352,Z 735.261,A 0.000,B 0.000,C 90.000,E1 82.996} C_DIS
LIN {X -0.063,Y -590.314,Z 735.254,A 0.000,B 0.000,C 90.000,E1 81.659} C_DIS
LIN {X 0.222,Y -590.182,Z 735.248,A 0.000,B 0.000,C 90.000,E1 80.566} C_DIS
LIN {X 0.115,Y -589.867,Z 735.242,A 0.000,B 0.000,C 90.000,E1 79.511} C_DIS
LIN {X 0.162,Y -589.328,Z 735.234,A 0.000,B 0.000,C 90.000,E1 78.173} C_DIS
LIN {X -0.006,Y -588.513,Z 735.226,A 0.000,B 0.000,C 90.000,E1 76.589} C_DIS
LIN {X 0.266,Y -587.732,Z 735.218,A 0.000,B 0.000,C 90.000,E1 75.227} C_DIS
LIN {X -0.042,Y -586.876,Z 735.211,A 0.000,B 0.000,C 90.000,E1 73.921} C_DIS
LIN {X 0.032,Y -585.642,Z 735.202,A 0.000,B 0.000,C 90.000,E1 72.308} C_DIS
LIN {X 0.038,Y -584.450,Z 735.194,A 0.000,B 0.000,C 90.000,E1 70.967} C_DIS
LIN {X 0.034,Y -583.186,Z 735.187,A 0.000,B 0.000,C 90.000,E1 69.625} C_DIS
LIN {X 0.002,Y -581.743,Z 735.179,A 0.000,B 0.000,C 90.000,E1 68.284} C_DIS
LIN {X -0.240,Y -580.389,Z 735.173,A 0.000,B 0.000,C 90.000,E1 67.230} C_DIS
LIN {X 0.261,Y -578.951,Z 735.167,A 0.000,B 0.000,C 90.000,E1 66.102} C_DIS
LIN {X -0.175,Y -576.841,Z 735.160,A 0.000,B 0.000,C 90.000,E1 64.793} C_DIS
LIN {X -0.001,Y -574.887,Z 735.154,A 0.000,B 0.000,C 90.000,E1 63.691} C_DIS
LIN {X -0.108,Y -572.715,Z 735.148,A 0.000,B 0.000,C 90.000,E1 62.615} C_DIS
LIN {X 0.177,Y -570.828,Z 735.143,A 0.000,B 0.000,C 90.000,E1 61.769} C_DIS
LIN {X -0.230,Y -568.018,Z 735.137,A 0.000,B 0.000,C 90.000,E1 60.717} C_DIS
LIN {X 0.004,Y -565.742,Z 735.133,A 0.000,B 0.000,C 90.000,E1 59.871} C_DIS
LIN {X -0.280,Y -563.204,Z 735.128,A 0.000,B 0.000,C 90.000,E1 59.076} C_DIS
LIN {X 0.182,Y -560.506,Z 735.123,A 0.000,B 0.000,C 90.000,E1 58.201} C_DIS
LIN {X 0.139,Y -557.538,Z 735.119,A 0.000,B 0.000,C 90.000,E1 57.375} C_DIS
LIN {X -0.005,Y -555.372,Z 735.116,A 0.000,B 0.000,C 90.000,E1 56.834} C_DIS
LIN {X -0.219,Y -551.107,Z 735.110,A 0.000,B 0.000,C 90.000,E1 55.881} C_DIS
LIN {X -0.102,Y -548.484,Z 735.107,A 0.000,B 0.000,C 90.000,E1 55.308} C_DIS
LIN {X -0.274,Y -544.054,Z 735.103,A 0.000,B 0.000,C 90.000,E1 54.482} C_DIS
LIN {X -0.032,Y -540.033,Z 735.099,A 0.000,B 0.000,C 90.000,E1 53.749} C_DIS
LIN {X -0.159,Y -537.525,Z 735.096,A 0.000,B 0.000,C 90.000,E1 53.336} C_DIS
LIN {X -0.136,Y -533.842,Z 735.093,A 0.000,B 0.000,C 90.000,E1 52.763} C_DIS
LIN {X -0.141,Y -529.695,Z 735.090,A 0.000,B 0.000,C 90.000,E1 52.190} C_DIS
LIN {X -0.177,Y -525.127,Z 735.087,A 0.000,B 0.000,C 90.000,E1 51.618} C_DIS
LIN {X 0.131,Y -519.932,Z 735.083,A 0.000,B 0.000,C 90.000,E1 51.009} C_DIS
LIN {X 0.110,Y -515.841,Z 735.081,A 0.000,B 0.000,C 90.000,E1 50.598} C_DIS
LIN {X 0.032,Y -510.400,Z 735.078,A 0.000,B 0.000,C 90.000,E1 50.114} C_DIS
LIN {X -0.107,Y -504.353,Z 735.076,A 0.000,B 0.000,C 90.000,E1 49.622} C_DIS
LIN {X 0.021,Y -498.030,Z 735.073,A 0.000,B 0.000,C 90.000,E1 49.138} C_DIS
LIN {X 0.145,Y -490.044,Z 735.070,A 0.000,B 0.000,C 90.000,E1 48.566} C_DIS
LIN {X -0.053,Y -483.415,Z 735.068,A 0.000,B 0.000,C 90.000,E1 48.162} C_DIS
LIN {X 0.246,Y -470.295,Z 735.063,A 0.000,B 0.000,C 90.000,E1 47.310} C_DIS
LIN {X 0.060,Y -452.537,Z 735.057,A 0.000,B 0.000,C 90.000,E1 46.215} C_DIS
LIN {X -0.167,Y -431.367,Z 735.049,A 0.000,B 0.000,C 90.000,E1 44.838} C_DIS
LIN {X -0.132,Y -423.425,Z 735.046,A 0.000,B 0.000,C 90.000,E1 44.271} C_DIS
LIN {X 0.201,Y -415.857,Z 735.043,A 0.000,B 0.000,C 90.000,E1 43.623} C_DIS
LIN {X 0.172,Y -415.830,Z 735.043,A 0.000,B 0.000,C 90.000,E1 43.623} C_DIS
LIN {X 0.054,Y -406.823,Z 735.017,A 0.000,B 0.000,C 90.000,E1 39.072} C_DIS
LIN {X 0.029,Y -405.647,Z 735.013,A 0.000,B 0.000,C 90.000,E1 38.382} C_DIS
LIN {X 0.015,Y -403.912,Z 735.009,A 0.000,B 0.000,C 90.000,E1 37.604} C_DIS
LIN {X -0.106,Y -403.874,Z 735.004,A 0.000,B 0.000,C 90.000,E1 36.664} C_DIS
LIN {X 0.116,Y -404.584,Z 734.986,A 0.000,B 0.000,C 90.000,E1 33.499} C_DIS
LIN {X -0.153,Y -405.272,Z 734.977,A 0.000,B 0.000,C 90.000,E1 31.799} C_DIS
LIN {X 0.101,Y -406.444,Z 734.963,A 0.000,B 0.000,C 90.000,E1 29.333} C_DIS
LIN {X -0.016,Y -407.764,Z 734.950,A 0.000,B 0.000,C 90.000,E1 26.924} C_DIS
LIN {X 0.011,Y -409.659,Z 734.934,A 0.000,B 0.000,C 90.000,E1 24.155} C_DIS
LIN {X -0.176,Y -412.723,Z 734.915,A 0.000,B 0.000,C 90.000,E1 20.737} C_DIS
LIN {X 0.037,Y -415.316,Z 734.902,A 0.000,B 0.000,C 90.000,E1 18.308} C_DIS
LIN {X 0.191,Y -418.362,Z 734.888,A 0.000,B 0.000,C 90.000,E1 15.898} C_DIS
LIN {X 0.085,Y -421.691,Z 734.875,A 0.000,B 0.000,C 90.000,E1 13.536} C_DIS
LIN {X -0.106,Y -424.718,Z 734.864,A 0.000,B 0.000,C 90.000,E1 11.535} C_DIS
LIN {X 0.022,Y -427.828,Z 734.853,A 0.000,B 0.000,C 90.000,E1 9.500} C_DIS
LIN {X 0.166,Y -430.884,Z 734.842,A 0.000,B 0.000,C 90.000,E1 7.473} C_DIS
LIN {X 0.019,Y -434.515,Z 734.829,A 0.000,B 0.000,C 90.000,E1 5.163} C_DIS
LIN {X -0.120,Y -438.388,Z 734.816,A 0.000,B 0.000,C 90.000,E1 2.865} C_DIS
LIN {X -0.195,Y -442.614,Z 734.803,A 0.000,B 0.000,C 90.000,E1 0.573} C_DIS
LIN {X -0.185,Y -446.570,Z 734.792,A 0.000,B 0.000,C 90.000,E1 358.511} C_DIS
LIN {X 0.169,Y -451.849,Z 734.777,A 0.000,B 0.000,C 90.000,E1 355.869} C_DIS
LIN {X -0.097,Y -456.091,Z 734.766,A 0.000,B 0.000,C 90.000,E1 353.970} C_DIS
LIN {X 0.003,Y -459.565,Z 734.758,A 0.000,B 0.000,C 90.000,E1 352.356} C_DIS
LIN {X 0.227,Y -463.004,Z 734.749,A 0.000,B 0.000,C 90.000,E1 350.735} C_DIS
LIN {X 0.135,Y -466.159,Z 734.740,A 0.000,B 0.000,C 90.000,E1 349.162} C_DIS
LIN {X -0.172,Y -468.582,Z 734.733,A 0.000,B 0.000,C 90.000,E1 347.937} C_DIS
LIN {X -0.136,Y -471.999,Z 734.722,A 0.000,B 0.000,C 90.000,E1 346.047} C_DIS
LIN {X -0.226,Y -476.658,Z 734.709,A 0.000,B 0.000,C 90.000,E1 343.559} C_DIS
LIN {X 0.006,Y -478.661,Z 734.703,A 0.000,B 0.000,C 90.000,E1 342.598} C_DIS
LIN {X 0.263,Y -481.115,Z 734.698,A 0.000,B 0.000,C 90.000,E1 341.638} C_DIS
LIN {X -0.133,Y -482.695,Z 734.696,A 0.000,B 0.000,C 90.000,E1 341.221} C_DIS
LIN {X 0.092,Y -484.858,Z 734.693,A 0.000,B 0.000,C 90.000,E1 340.732} C_DIS
LIN {X -0.215,Y -487.191,Z 734.691,A 0.000,B 0.000,C 90.000,E1 340.369} C_DIS
LIN {X 0.038,Y -490.665,Z 734.688,A 0.000,B 0.000,C 90.000,E1 339.880} C_DIS
LIN {X 0.077,Y -493.968,Z 734.686,A 0.000,B 0.000,C 90.000,E1 339.518} C_DIS
LIN {X -0.238,Y -500.190,Z 734.683,A 0.000,B 0.000,C 90.000,E1 339.028} C_DIS
LIN {X -0.202,Y -511.146,Z 734.679,A 0.000,B 0.000,C 90.000,E1 338.284} C_DIS
LIN {X -0.275,Y -533.540,Z 734.672,A 0.000,B 0.000,C 90.000,E1 336.922} C_DIS
LIN {X -0.058,Y -541.223,Z 734.669,A 0.000,B 0.000,C 90.000,E1 336.410} C_DIS
LIN {X -0.051,Y -547.062,Z 734.667,A 0.000,B 0.000,C 90.000,E1 335.973} C_DIS
LIN {X -0.076,Y -553.878,Z 734.663,A 0.000,B 0.000,C 90.000,E1 335.409} C_DIS
LIN {X -0.122,Y -559.154,Z 734.661,A 0.000,B 0.000,C 90.000,E1 334.921} C_DIS
LIN {X -0.168,Y -563.219,Z 734.659,A 0.000,B 0.000,C 90.000,E1 334.537} C_DIS
LIN {X -0.173,Y -570.612,Z 734.654,A 0.000,B 0.000,C 90.000,E1 333.768} C_DIS
LIN {X 0.018,Y -576.764,Z 734.651,A 0.000,B 0.000,C 90.000,E1 333.076} C_DIS
LIN {X -0.085,Y -582.550,Z 734.647,A 0.000,B 0.000,C 90.000,E1 332.410} C_DIS
LIN {X 0.134,Y -588.071,Z 734.643,A 0.000,B 0.000,C 90.000,E1 331.719} C_DIS
LIN {X 0.137,Y -593.440,Z 734.639,A 0.000,B 0.000,C 90.000,E1 331.051} C_DIS
LIN {X 0.150,Y -599.575,Z 734.635,A 0.000,B 0.000,C 90.000,E1 330.255} C_DIS
LIN {X 0.164,Y -607.373,Z 734.629,A 0.000,B 0.000,C 90.000,E1 329.203} C_DIS
LIN {X -0.180,Y -611.984,Z 734.625,A 0.000,B 0.000,C 90.000,E1 328.584} C_DIS
LIN {X 0.006,Y -618.128,Z 734.620,A 0.000,B 0.000,C 90.000,E1 327.661} C_DIS
LIN {X 0.065,Y -624.713,Z 734.615,A 0.000,B 0.000,C 90.000,E1 326.628} C_DIS
LIN {X -0.133,Y -628.549,Z 734.611,A 0.000,B 0.000,C 90.000,E1 326.008} C_DIS
LIN {X 0.064,Y -633.767,Z 734.606,A 0.000,B 0.000,C 90.000,E1 325.102} C_DIS
LIN {X -0.180,Y -639.944,Z 734.600,A 0.000,B 0.000,C 90.000,E1 323.989} C_DIS
LIN {X 0.131,Y -643.860,Z 734.596,A 0.000,B 0.000,C 90.000,E1 323.210} C_DIS
LIN {X -0.034,Y -647.579,Z 734.592,A 0.000,B 0.000,C 90.000,E1 322.477} C_DIS
LIN {X 0.278,Y -652.211,Z 734.586,A 0.000,B 0.000,C 90.000,E1 321.457} C_DIS
LIN {X 0.194,Y -655.541,Z 734.582,A 0.000,B 0.000,C 90.000,E1 320.723} C_DIS
LIN {X 0.103,Y -659.731,Z 734.576,A 0.000,B 0.000,C 90.000,E1 319.747} C_DIS
LIN {X 0.064,Y -663.703,Z 734.571,A 0.000,B 0.000,C 90.000,E1 318.771} C_DIS
LIN {X 0.070,Y -667.432,Z 734.566,A 0.000,B 0.000,C 90.000,E1 317.796} C_DIS
LIN {X 0.093,Y -671.547,Z 734.559,A 0.000,B 0.000,C 90.000,E1 316.581} C_DIS
LIN {X -0.276,Y -675.388,Z 734.552,A 0.000,B 0.000,C 90.000,E1 315.405} C_DIS
LIN {X -0.152,Y -678.252,Z 734.547,A 0.000,B 0.000,C 90.000,E1 314.433} C_DIS
LIN {X 0.049,Y -681.566,Z 734.540,A 0.000,B 0.000,C 90.000,E1 313.218} C_DIS
LIN {X -0.224,Y -683.981,Z 734.535,A 0.000,B 0.000,C 90.000,E1 312.285} C_DIS
LIN {X 0.047,Y -686.306,Z 734.530,A 0.000,B 0.000,C 90.000,E1 311.310} C_DIS
LIN {X -0.228,Y -687.915,Z 734.526,A 0.000,B 0.000,C 90.000,E1 310.620} C_DIS
LIN {X 0.099,Y -689.769,Z 734.520,A 0.000,B 0.000,C 90.000,E1 309.644} C_DIS
LIN {X -0.152,Y -690.988,Z 734.516,A 0.000,B 0.000,C 90.000,E1 308.955} C_DIS
LIN {X -0.227,Y -692.432,Z 734.511,A 0.000,B 0.000,C 90.000,E1 308.016} C_DIS
LIN {X 0.335,Y -693.979,Z 734.505,A 0.000,B 0.000,C 90.000,E1 306.790} C_DIS
LIN {X -0.109,Y -695.074,Z 734.499,A 0.000,B 0.000,C 90.000,E1 305.884} C_DIS
LIN {X -0.135,Y -696.010,Z 734.494,A 0.000,B 0.000,C 90.000,E1 304.945} C_DIS
LIN {X -0.322,Y -696.968,Z 734.488,A 0.000,B 0.000,C 90.000,E1 303.785} C_DIS
LIN {X -0.207,Y -698.340,Z 734.478,A 0.000,B 0.000,C 90.000,E1 302.133} C_DIS
LIN {X 0.237,Y -699.282,Z 734.472,A 0.000,B 0.000,C 90.000,E1 300.924} C_DIS
LIN {X 0.077,Y -699.741,Z 734.467,A 0.000,B 0.000,C 90.000,E1 300.001} C_DIS
LIN {X 0.194,Y -700.068,Z 734.460,A 0.000,B 0.000,C 90.000,E1 298.821} C_DIS
LIN {X 0.188,Y -700.631,Z 734.450,A 0.000,B 0.000,C 90.000,E1 296.950} C_DIS
LIN {X -0.085,Y -701.372,Z 734.441,A 0.000,B 0.000,C 90.000,E1 295.335} C_DIS
LIN {X -0.194,Y -701.361,Z 734.437,A 0.000,B 0.000,C 90.000,E1 294.643} C_DIS
LIN {X 0.079,Y -700.953,Z 734.436,A 0.000,B 0.000,C 90.000,E1 294.387} C_DIS
LIN {X -0.302,Y -699.650,Z 734.433,A 0.000,B 0.000,C 90.000,E1 293.951} C_DIS
LIN {X -0.167,Y -699.070,Z 734.432,A 0.000,B 0.000,C 90.000,E1 293.823} C_DIS
LIN {X 0.097,Y -697.171,Z 734.431,A 0.000,B 0.000,C 90.000,E1 293.567} C_DIS
LIN {X 0.207,Y -693.719,Z 734.429,A 0.000,B 0.000,C 90.000,E1 293.206} C_DIS
LIN {X 0.339,Y -692.091,Z 734.428,A 0.000,B 0.000,C 90.000,E1 293.078} C_DIS
LIN {X 0.231,Y -687.680,Z 734.427,A 0.000,B 0.000,C 90.000,E1 292.898} C_DIS
LIN {X 0.261,Y -685.821,Z 734.427,A 0.000,B 0.000,C 90.000,E1 292.823} C_DIS
LIN {X -0.035,Y -681.562,Z 734.426,A 0.000,B 0.000,C 90.000,E1 292.717} C_DIS
LIN {X 0.223,Y -677.329,Z 734.426,A 0.000,B 0.000,C 90.000,E1 292.589} C_DIS
LIN {X -0.295,Y -674.898,Z 734.425,A 0.000,B 0.000,C 90.000,E1 292.589} C_DIS
LIN {X 0.129,Y -668.121,Z 734.425,A 0.000,B 0.000,C 90.000,E1 292.461} C_DIS
LIN {X -0.064,Y -660.244,Z 734.424,A 0.000,B 0.000,C 90.000,E1 292.386} C_DIS
LIN {X 0.231,Y -646.734,Z 734.423,A 0.000,B 0.000,C 90.000,E1 292.153} C_DIS
LIN {X 0.190,Y -633.344,Z 734.422,A 0.000,B 0.000,C 90.000,E1 291.897} C_DIS
LIN {X -0.329,Y -623.602,Z 734.421,A 0.000,B 0.000,C 90.000,E1 291.716} C_DIS
LIN {X 0.006,Y -599.568,Z 734.417,A 0.000,B 0.000,C 90.000,E1 291.046} C_DIS
LIN {X 0.089,Y -578.456,Z 734.414,A 0.000,B 0.000,C 90.000,E1 290.429} C_DIS
LIN {X -0.136,Y -571.065,Z 734.412,A 0.000,B 0.000,C 90.000,E1 290.248} C_DIS
LIN {X 0.202,Y -567.429,Z 734.412,A 0.000,B 0.000,C 90.000,E1 290.120} C_DIS
LIN {X 0.159,Y -562.039,Z 734.411,A 0.000,B 0.000,C 90.000,E1 289.939} C_DIS
LIN {X 0.096,Y -560.599,Z 734.411,A 0.000,B 0.000,C 90.000,E1 289.885} C_DIS
LIN {X -0.175,Y -556.724,Z 734.409,A 0.000,B 0.000,C 90.000,E1 289.685} C_DIS
LIN {X 0.294,Y -556.642,Z 734.409,A 0.000,B 0.000,C 90.000,E1 289.631} C_DIS
LIN {X 0.251,Y -555.585,Z 734.408,A 0.000,B 0.000,C 90.000,E1 289.450} C_DIS
LIN {X 0.052,Y -554.933,Z 734.406,A 0.000,B 0.000,C 90.000,E1 289.087} C_DIS
LIN {X -0.059,Y -554.309,Z 734.397,A 0.000,B 0.000,C 90.000,E1 287.511} C_DIS
LIN {X 0.296,Y -553.825,Z 734.390,A 0.000,B 0.000,C 90.000,E1 286.079} C_DIS
LIN {X 0.083,Y -553.173,Z 734.380,A 0.000,B 0.000,C 90.000,E1 284.426} C_DIS
LIN {X -0.256,Y -552.758,Z 734.372,A 0.000,B 0.000,C 90.000,E1 283.063} C_DIS
LIN {X -0.071,Y -552.203,Z 734.363,A 0.000,B 0.000,C 90.000,E1 281.366} C_DIS
LIN {X -0.019,Y -551.643,Z 734.355,A 0.000,B 0.000,C 90.000,E1 279.962} C_DIS
LIN {X -0.081,Y -550.962,Z 734.348,A 0.000,B 0.000,C 90.000,E1 278.568} C_DIS
LIN {X -0.130,Y -550.183,Z 734.338,A 0.000,B 0.000,C 90.000,E1 276.891} C_DIS
LIN {X -0.261,Y -549.474,Z 734.329,A 0.000,B 0.000,C 90.000,E1 275.220} C_DIS
LIN {X -0.034,Y -549.018,Z 734.323,A 0.000,B 0.000,C 90.000,E1 274.073} C_DIS
LIN {X -0.181,Y -548.079,Z 734.312,A 0.000,B 0.000,C 90.000,E1 272.121} C_DIS
LIN {X -0.022,Y -547.705,Z 734.307,A 0.000,B 0.000,C 90.000,E1 271.260} C_DIS
LIN {X 0.257,Y -546.734,Z 734.298,A 0.000,B 0.000,C 90.000,E1 269.542} C_DIS
LIN {X -0.020,Y -545.669,Z 734.288,A 0.000,B 0.000,C 90.000,E1 267.879} C_DIS
LIN {X 0.222,Y -544.574,Z 734.279,A 0.000,B 0.000,C 90.000,E1 266.159} C_DIS
LIN {X -0.102,Y -543.637,Z 734.271,A 0.000,B 0.000,C 90.000,E1 264.780} C_DIS
LIN {X 0.155,Y -542.584,Z 734.263,A 0.000,B 0.000,C 90.000,E1 263.337} C_DIS
LIN {X -0.217,Y -541.725,Z 734.257,A 0.000,B 0.000,C 90.000,E1 262.243} C_DIS
LIN {X 0.136,Y -540.052,Z 734.246,A 0.000,B 0.000,C 90.000,E1 260.218} C_DIS
LIN {X 0.031,Y -538.607,Z 734.236,A 0.000,B 0.000,C 90.000,E1 258.522} C_DIS
LIN {X -0.162,Y -537.461,Z 734.228,A 0.000,B 0.000,C 90.000,E1 257.117} C_DIS
LIN {X 0.205,Y -536.461,Z 734.222,A 0.000,B 0.000,C 90.000,E1 255.936} C_DIS
LIN {X 0.282,Y -534.624,Z 734.213,A 0.000,B 0.000,C 90.000,E1 254.212} C_DIS
LIN {X -0.197,Y -532.805,Z 734.203,A 0.000,B 0.000,C 90.000,E1 252.543} C_DIS
LIN {X -0.076,Y -531.250,Z 734.195,A 0.000,B 0.000,C 90.000,E1 251.094} C_DIS
LIN {X 0.006,Y -529.720,Z 734.189,A 0.000,B 0.000,C 90.000,E1 249.934} C_DIS
LIN {X 0.247,Y -527.793,Z 734.181,A 0.000,B 0.000,C 90.000,E1 248.465} C_DIS
LIN {X 0.095,Y -526.553,Z 734.176,A 0.000,B 0.000,C 90.000,E1 247.614} C_DIS
LIN {X -0.021,Y -524.378,Z 734.168,A 0.000,B 0.000,C 90.000,E1 246.177} C_DIS
LIN {X -0.014,Y -523.003,Z 734.163,A 0.000,B 0.000,C 90.000,E1 245.305} C_DIS
LIN {X 0.021,Y -520.633,Z 734.155,A 0.000,B 0.000,C 90.000,E1 243.845} C_DIS
LIN {X 0.114,Y -518.573,Z 734.148,A 0.000,B 0.000,C 90.000,E1 242.666} C_DIS
LIN {X 0.306,Y -515.704,Z 734.140,A 0.000,B 0.000,C 90.000,E1 241.179} C_DIS
LIN {X -0.108,Y -512.260,Z 734.130,A 0.000,B 0.000,C 90.000,E1 239.459} C_DIS
LIN {X -0.233,Y -509.276,Z 734.122,A 0.000,B 0.000,C 90.000,E1 237.995} C_DIS
LIN {X -0.149,Y -506.115,Z 734.114,A 0.000,B 0.000,C 90.000,E1 236.501} C_DIS
LIN {X -0.043,Y -504.209,Z 734.109,A 0.000,B 0.000,C 90.000,E1 235.595} C_DIS
LIN {X -0.073,Y -501.422,Z 734.102,A 0.000,B 0.000,C 90.000,E1 234.402} C_DIS
LIN {X -0.146,Y -498.543,Z 734.096,A 0.000,B 0.000,C 90.000,E1 233.210} C_DIS
LIN {X 0.062,Y -493.902,Z 734.086,A 0.000,B 0.000,C 90.000,E1 231.376} C_DIS
LIN {X 0.166,Y -489.544,Z 734.075,A 0.000,B 0.000,C 90.000,E1 229.542} C_DIS
LIN {X 0.252,Y -484.645,Z 734.063,A 0.000,B 0.000,C 90.000,E1 227.391} C_DIS
LIN {X -0.072,Y -481.292,Z 734.055,A 0.000,B 0.000,C 90.000,E1 225.891} C_DIS
LIN {X 0.110,Y -476.610,Z 734.043,A 0.000,B 0.000,C 90.000,E1 223.704} C_DIS
LIN {X 0.086,Y -472.675,Z 734.033,A 0.000,B 0.000,C 90.000,E1 221.838} C_DIS
LIN {X -0.188,Y -469.938,Z 734.026,A 0.000,B 0.000,C 90.000,E1 220.620} C_DIS
LIN {X 0.044,Y -465.774,Z 734.015,A 0.000,B 0.000,C 90.000,E1 218.705} C_DIS
LIN {X -0.225,Y -462.273,Z 734.006,A 0.000,B 0.000,C 90.000,E1 217.156} C_DIS
LIN {X 0.169,Y -458.976,Z 733.997,A 0.000,B 0.000,C 90.000,E1 215.518} C_DIS
LIN {X -0.125,Y -453.372,Z 733.982,A 0.000,B 0.000,C 90.000,E1 212.673} C_DIS
LIN {X 0.122,Y -449.200,Z 733.969,A 0.000,B 0.000,C 90.000,E1 210.384} C_DIS
LIN {X 0.192,Y -444.981,Z 733.956,A 0.000,B 0.000,C 90.000,E1 208.103} C_DIS
LIN {X 0.098,Y -441.330,Z 733.945,A 0.000,B 0.000,C 90.000,E1 206.155} C_DIS
LIN {X -0.071,Y -437.690,Z 733.935,A 0.000,B 0.000,C 90.000,E1 204.207} C_DIS
LIN {X 0.077,Y -433.981,Z 733.923,A 0.000,B 0.000,C 90.000,E1 202.206} C_DIS
LIN {X -0.188,Y -430.268,Z 733.912,A 0.000,B 0.000,C 90.000,E1 200.248} C_DIS
LIN {X -0.141,Y -427.817,Z 733.905,A 0.000,B 0.000,C 90.000,E1 198.906} C_DIS
LIN {X 0.135,Y -425.340,Z 733.898,A 0.000,B 0.000,C 90.000,E1 197.528} C_DIS
LIN {X 0.150,Y -422.070,Z 733.888,A 0.000,B 0.000,C 90.000,E1 195.843} C_DIS
LIN {X 0.089,Y -417.730,Z 733.875,A 0.000,B 0.000,C 90.000,E1 193.480} C_DIS
LIN {X 0.130,Y -414.773,Z 733.866,A 0.000,B 0.000,C 90.000,E1 191.771} C_DIS
LIN {X 0.116,Y -409.962,Z 733.850,A 0.000,B 0.000,C 90.000,E1 189.029} C_DIS
LIN {X 0.154,Y -406.067,Z 733.837,A 0.000,B 0.000,C 90.000,E1 186.606} C_DIS
LIN {X 0.091,Y -402.917,Z 733.825,A 0.000,B 0.000,C 90.000,E1 184.531} C_DIS
LIN {X 0.155,Y -398.628,Z 733.808,A 0.000,B 0.000,C 90.000,E1 181.375} C_DIS
LIN {X -0.058,Y -396.928,Z 733.800,A 0.000,B 0.000,C 90.000,E1 180.000} C_DIS
LIN {X 0.100,Y -395.493,Z 733.792,A 0.000,B 0.000,C 90.000,E1 178.568} C_DIS
LIN {X 0.190,Y -393.743,Z 733.782,A 0.000,B 0.000,C 90.000,E1 176.788} C_DIS
LIN {X -0.133,Y -390.443,Z 733.761,A 0.000,B 0.000,C 90.000,E1 172.932} C_DIS
LIN {X 0.039,Y -388.649,Z 733.741,A 0.000,B 0.000,C 90.000,E1 169.342} C_DIS
LIN {X -0.125,Y -388.059,Z 733.733,A 0.000,B 0.000,C 90.000,E1 167.937} C_DIS
LIN {X 0.120,Y -387.303,Z 733.721,A 0.000,B 0.000,C 90.000,E1 165.755} C_DIS
LIN {X 0.022,Y -386.897,Z 733.713,A 0.000,B 0.000,C 90.000,E1 164.338} C_DIS
LIN {X 0.097,Y -386.489,Z 733.699,A 0.000,B 0.000,C 90.000,E1 161.819} C_DIS
LIN {X -0.136,Y -386.190,Z 733.689,A 0.000,B 0.000,C 90.000,E1 160.061} C_DIS
LIN {X -0.061,Y -385.918,Z 733.675,A 0.000,B 0.000,C 90.000,E1 157.539} C_DIS
LIN {X 0.132,Y -385.787,Z 733.657,A 0.000,B 0.000,C 90.000,E1 154.280} C_DIS
LIN {X 0.135,Y -386.462,Z 733.639,A 0.000,B 0.000,C 90.000,E1 151.051} C_DIS
LIN {X 0.028,Y -387.707,Z 733.623,A 0.000,B 0.000,C 90.000,E1 148.201} C_DIS
LIN {X -0.186,Y -389.197,Z 733.612,A 0.000,B 0.000,C 90.000,E1 146.087} C_DIS
LIN {X -0.004,Y -392.159,Z 733.596,A 0.000,B 0.000,C 90.000,E1 143.210} C_DIS
LIN {X -0.003,Y -393.558,Z 733.590,A 0.000,B 0.000,C 90.000,E1 142.145} C_DIS
LIN {X 0.040,Y -395.682,Z 733.582,A 0.000,B 0.000,C 90.000,E1 140.723} C_DIS
LIN {X -0.074,Y -397.069,Z 733.578,A 0.000,B 0.000,C 90.000,E1 140.033} C_DIS
LIN {X 0.029,Y -399.181,Z 733.573,A 0.000,B 0.000,C 90.000,E1 139.138} C_DIS
LIN {X -0.180,Y -401.742,Z 733.569,A 0.000,B 0.000,C 90.000,E1 138.405} C_DIS
LIN {X 0.004,Y -403.554,Z 733.567,A 0.000,B 0.000,C 90.000,E1 138.000} C_DIS
LIN {X -0.086,Y -404.279,Z 733.566,A 0.000,B 0.000,C 90.000,E1 137.838} C_DIS
LIN {X -0.043,Y -407.498,Z 733.563,A 0.000,B 0.000,C 90.000,E1 137.310} C_DIS
LIN {X -0.146,Y -411.672,Z 733.560,A 0.000,B 0.000,C 90.000,E1 136.782} C_DIS
LIN {X 0.051,Y -418.896,Z 733.555,A 0.000,B 0.000,C 90.000,E1 135.972} C_DIS
LIN {X -0.085,Y -433.798,Z 733.547,A 0.000,B 0.000,C 90.000,E1 134.514} C_DIS
LIN {X 0.161,Y -447.100,Z 733.540,A 0.000,B 0.000,C 90.000,E1 133.218} C_DIS
LIN {X -0.015,Y -455.927,Z 733.536,A 0.000,B 0.000,C 90.000,E1 132.405} C_DIS
LIN {X -0.075,Y -467.102,Z 733.529,A 0.000,B 0.000,C 90.000,E1 131.310} C_DIS
LIN {X -0.148,Y -476.791,Z 733.524,A 0.000,B 0.000,C 90.000,E1 130.334} C_DIS
LIN {X 0.107,Y -480.842,Z 733.522,A 0.000,B 0.000,C 90.000,E1 129.886} C_DIS
LIN {X 0.049,Y -488.827,Z 733.517,A 0.000,B 0.000,C 90.000,E1 129.036} C_DIS
LIN {X 0.001,Y -495.076,Z 733.513,A 0.000,B 0.000,C 90.000,E1 128.338} C_DIS
LIN {X 0.065,Y -498.831,Z 733.511,A 0.000,B 0.000,C 90.000,E1 127.890} C_DIS
LIN {X -0.066,Y -503.474,Z 733.507,A 0.000,B 0.000,C 90.000,E1 127.317} C_DIS
LIN {X 0.015,Y -507.842,Z 733.504,A 0.000,B 0.000,C 90.000,E1 126.710} C_DIS
LIN {X -0.091,Y -512.010,Z 733.501,A 0.000,B 0.000,C 90.000,E1 126.137} C_DIS
LIN {X 0.161,Y -515.943,Z 733.497,A 0.000,B 0.000,C 90.000,E1 125.518} C_DIS
LIN {X 0.023,Y -519.510,Z 733.494,A 0.000,B 0.000,C 90.000,E1 124.945} C_DIS
LIN {X 0.165,Y -523.645,Z 733.490,A 0.000,B 0.000,C 90.000,E1 124.199} C_DIS
LIN {X -0.085,Y -527.382,Z 733.486,A 0.000,B 0.000,C 90.000,E1 123.499} C_DIS
LIN {X 0.293,Y -530.219,Z 733.483,A 0.000,B 0.000,C 90.000,E1 122.880} C_DIS
LIN {X -0.059,Y -534.114,Z 733.478,A 0.000,B 0.000,C 90.000,E1 122.054} C_DIS
LIN {X 0.120,Y -539.581,Z 733.471,A 0.000,B 0.000,C 90.000,E1 120.747} C_DIS
LIN {X 0.058,Y -544.091,Z 733.465,A 0.000,B 0.000,C 90.000,E1 119.617} C_DIS
LIN {X 0.301,Y -547.357,Z 733.460,A 0.000,B 0.000,C 90.000,E1 118.743} C_DIS
LIN {X 0.074,Y -551.452,Z 733.454,A 0.000,B 0.000,C 90.000,E1 117.641} C_DIS
LIN {X -0.101,Y -555.108,Z 733.447,A 0.000,B 0.000,C 90.000,E1 116.539} C_DIS
LIN {X -0.260,Y -557.478,Z 733.443,A 0.000,B 0.000,C 90.000,E1 115.720} C_DIS
LIN {X 0.117,Y -559.543,Z 733.438,A 0.000,B 0.000,C 90.000,E1 114.847} C_DIS
LIN {X 0.012,Y -561.371,Z 733.434,A 0.000,B 0.000,C 90.000,E1 114.027} C_DIS
LIN {X -0.077,Y -562.924,Z 733.429,A 0.000,B 0.000,C 90.000,E1 113.206} C_DIS
LIN {X -0.240,Y -565.066,Z 733.421,A 0.000,B 0.000,C 90.000,E1 111.844} C_DIS
LIN {X -0.037,Y -567.565,Z 733.412,A 0.000,B 0.000,C 90.000,E1 110.174} C_DIS
LIN {X -0.136,Y -569.173,Z 733.406,A 0.000,B 0.000,C 90.000,E1 109.087} C_DIS
LIN {X -0.239,Y -571.329,Z 733.397,A 0.000,B 0.000,C 90.000,E1 107.457} C_DIS
LIN {X -0.125,Y -573.675,Z 733.386,A 0.000,B 0.000,C 90.000,E1 105.536} C_DIS
LIN {X -0.097,Y -574.652,Z 733.382,A 0.000,B 0.000,C 90.000,E1 104.717} C_DIS
LIN {X -0.058,Y -576.279,Z 733.374,A 0.000,B 0.000,C 90.000,E1 103.355} C_DIS
LIN {X 0.090,Y -578.227,Z 733.365,A 0.000,B 0.000,C 90.000,E1 101.715} C_DIS
LIN {X 0.054,Y -579.873,Z 733.358,A 0.000,B 0.000,C 90.000,E1 100.366} C_DIS
LIN {X 0.054,Y -580.823,Z 733.353,A 0.000,B 0.000,C 90.000,E1 99.557} C_DIS
LIN {X -0.278,Y -581.991,Z 733.347,A 0.000,B 0.000,C 90.000,E1 98.511} C_DIS
LIN {X 0.133,Y -583.286,Z 733.340,A 0.000,B 0.000,C 90.000,E1 97.125} C_DIS
LIN {X -0.013,Y -584.593,Z 733.332,A 0.000,B 0.000,C 90.000,E1 95.796} C_DIS
LIN {X -0.202,Y -585.850,Z 733.325,A 0.000,B 0.000,C 90.000,E1 94.473} C_DIS
LIN {X 0.212,Y -587.019,Z 733.317,A 0.000,B 0.000,C 90.000,E1 93.094} C_DIS
LIN {X 0.020,Y -588.023,Z 733.310,A 0.000,B 0.000,C 90.000,E1 91.776} C_DIS
LIN {X 0.034,Y -589.008,Z 733.301,A 0.000,B 0.000,C 90.000,E1 90.172} C_DIS
LIN {X -0.133,Y -589.679,Z 733.294,A 0.000,B 0.000,C 90.000,E1 88.854} C_DIS
LIN {X 0.129,Y -590.327,Z 733.283,A 0.000,B 0.000,C 90.000,E1 86.963} C_DIS
LIN {X 0.031,Y -590.599,Z 733.276,A 0.000,B 0.000,C 90.000,E1 85.641} C_DIS
LIN {X -0.055,Y -590.775,Z 733.268,A 0.000,B 0.000,C 90.000,E1 84.318} C_DIS
LIN {X -0.147,Y -590.864,Z 733.261,A 0.000,B 0.000,C 90.000,E1 82.996} C_DIS
LIN {X -0.089,Y -590.816,Z 733.254,A 0.000,B 0.000,C 90.000,E1 81.659} C_DIS
LIN {X -0.114,Y -590.598,Z 733.246,A 0.000,B 0.000,C 90.000,E1 80.330} C_DIS
LIN {X -0.210,Y -590.231,Z 733.240,A 0.000,B 0.000,C 90.000,E1 79.275} C_DIS
LIN {X 0.157,Y -589.768,Z 733.234,A 0.000,B 0.000,C 90.000,E1 78.173} C_DIS
LIN {X -0.002,Y -588.914,Z 733.226,A 0.000,B 0.000,C 90.000,E1 76.589} C_DIS
LIN {X 0.277,Y -588.123,Z 733.218,A 0.000,B 0.000,C 90.000,E1 75.227} C_DIS
LIN {X -0.025,Y -587.221,Z 733.211,A 0.000,B 0.000,C 90.000,E1 73.921} C_DIS
LIN {X 0.057,Y -585.961,Z 733.202,A 0.000,B 0.000,C 90.000,E1 72.308} C_DIS
LIN {X -0.266,Y -584.479,Z 733.193,A 0.000,B 0.000,C 90.000,E1 70.732} C_DIS
LIN {X 0.069,Y -583.443,Z 733.187,A 0.000,B 0.000,C 90.000,E1 69.625} C_DIS
LIN {X 0.042,Y -581.956,Z 733.179,A 0.000,B 0.000,C 90.000,E1 68.284} C_DIS
LIN {X -0.197,Y -580.578,Z 733.173,A 0.000,B 0.000,C 90.000,E1 67.230} C_DIS
LIN {X 0.306,Y -579.098,Z 733.167,A 0.000,B 0.000,C 90.000,E1 66.102} C_DIS
LIN {X 0.019,Y -577.368,Z 733.161,A 0.000,B 0.000,C 90.000,E1 65.049} C_DIS
LIN {X -0.055,Y -575.485,Z 733.155,A 0.000,B 0.000,C 90.000,E1 63.973} C_DIS
LIN {X -0.060,Y -572.724,Z 733.148,A 0.000,B 0.000,C 90.000,E1 62.615} C_DIS
LIN {X 0.059,Y -570.079,Z 733.142,A 0.000,B 0.000,C 90.000,E1 61.513} C_DIS
LIN {X -0.182,Y -567.926,Z 733.137,A 0.000,B 0.000,C 90.000,E1 60.717} C_DIS
LIN {X 0.050,Y -565.617,Z 733.133,A 0.000,B 0.000,C 90.000,E1 59.871} C_DIS
LIN {X -0.141,Y -562.095,Z 733.127,A 0.000,B 0.000,C 90.000,E1 58.791} C_DIS
LIN {X 0.224,Y -560.289,Z 733.124,A 0.000,B 0.000,C 90.000,E1 58.201} C_DIS
LIN {X 0.180,Y -557.249,Z 733.119,A 0.000,B 0.000,C 90.000,E1 57.375} C_DIS
LIN {X 0.034,Y -555.029,Z 733.116,A 0.000,B 0.000,C 90.000,E1 56.834} C_DIS
LIN {X -0.188,Y -550.666,Z 733.110,A 0.000,B 0.000,C 90.000,E1 55.881} C_DIS
LIN {X -0.074,Y -548.008,Z 733.107,A 0.000,B 0.000,C 90.000,E1 55.308} C_DIS
LIN {X -0.178,Y -543.470,Z 733.103,A 0.000,B 0.000,C 90.000,E1 54.482} C_DIS
LIN {X -0.112,Y -540.235,Z 733.099,A 0.000,B 0.000,C 90.000,E1 53.909} C_DIS
LIN {X -0.023,Y -536.816,Z 733.096,A 0.000,B 0.000,C 90.000,E1 53.336} C_DIS
LIN {X -0.007,Y -533.014,Z 733.093,A 0.000,B 0.000,C 90.000,E1 52.763} C_DIS
LIN {X -0.019,Y -528.784,Z 733.090,A 0.000,B 0.000,C 90.000,E1 52.190} C_DIS
LIN {X -0.036,Y -524.047,Z 733.087,A 0.000,B 0.000,C 90.000,E1 51.618} C_DIS
LIN {X 0.152,Y -520.157,Z 733.084,A 0.000,B 0.000,C 90.000,E1 51.170} C_DIS
LIN {X 0.188,Y -514.903,Z 733.081,A 0.000,B 0.000,C 90.000,E1 50.642} C_DIS
LIN {X -0.082,Y -508.929,Z 733.079,A 0.000,B 0.000,C 90.000,E1 50.150} C_DIS
LIN {X 0.205,Y -504.514,Z 733.077,A 0.000,B 0.000,C 90.000,E1 49.747} C_DIS
LIN {X 0.161,Y -496.591,Z 733.073,A 0.000,B 0.000,C 90.000,E1 49.175} C_DIS
LIN {X -0.162,Y -490.158,Z 733.071,A 0.000,B 0.000,C 90.000,E1 48.771} C_DIS
LIN {X 0.234,Y -485.246,Z 733.069,A 0.000,B 0.000,C 90.000,E1 48.405} C_DIS
LIN {X -0.122,Y -472.140,Z 733.065,A 0.000,B 0.000,C 90.000,E1 47.634} C_DIS
LIN {X -0.104,Y -455.997,Z 733.059,A 0.000,B 0.000,C 90.000,E1 46.620} C_DIS
LIN {X 0.047,Y -431.643,Z 733.050,A 0.000,B 0.000,C 90.000,E1 45.000} C_DIS
LIN {X 0.042,Y -425.232,Z 733.048,A 0.000,B 0.000,C 90.000,E1 44.555} C_DIS
LIN {X -0.019,Y -416.358,Z 733.044,A 0.000,B 0.000,C 90.000,E1 43.866} C_DIS
LIN {X -0.048,Y -416.326,Z 733.044,A 0.000,B 0.000,C 90.000,E1 43.866} C_DIS
LIN {X -0.195,Y -406.971,Z 733.018,A 0.000,B 0.000,C 90.000,E1 39.197} C_DIS
LIN {X 0.097,Y -405.845,Z 733.014,A 0.000,B 0.000,C 90.000,E1 38.463} C_DIS
LIN {X 0.085,Y -404.160,Z 733.009,A 0.000,B 0.000,C 90.000,E1 37.684} C_DIS
LIN {X -0.153,Y -404.724,Z 732.991,A 0.000,B 0.000,C 90.000,E1 34.326} C_DIS
LIN {X -0.049,Y -405.645,Z 732.977,A 0.000,B 0.000,C 90.000,E1 31.878} C_DIS
LIN {X -0.133,Y -406.791,Z 732.964,A 0.000,B 0.000,C 90.000,E1 29.461} C_DIS
LIN {X -0.151,Y -407.927,Z 732.952,A 0.000,B 0.000,C 90.000,E1 27.385} C_DIS
LIN {X 0.044,Y -409.209,Z 732.941,A 0.000,B 0.000,C 90.000,E1 25.283} C_DIS
LIN {X -0.157,Y -411.130,Z 732.927,A 0.000,B 0.000,C 90.000,E1 22.898} C_DIS
LIN {X 0.159,Y -413.044,Z 732.916,A 0.000,B 0.000,C 90.000,E1 20.791} C_DIS
LIN {X -0.164,Y -415.226,Z 732.904,A 0.000,B 0.000,C 90.000,E1 18.779} C_DIS
LIN {X 0.223,Y -417.727,Z 732.893,A 0.000,B 0.000,C 90.000,E1 16.677} C_DIS
LIN {X -0.014,Y -419.979,Z 732.883,A 0.000,B 0.000,C 90.000,E1 15.009} C_DIS
LIN {X 0.026,Y -421.934,Z 732.876,A 0.000,B 0.000,C 90.000,E1 13.647} C_DIS
LIN {X 0.165,Y -424.926,Z 732.865,A 0.000,B 0.000,C 90.000,E1 11.602} C_DIS
LIN {X -0.039,Y -428.016,Z 732.853,A 0.000,B 0.000,C 90.000,E1 9.613} C_DIS
LIN {X 0.105,Y -431.051,Z 732.842,A 0.000,B 0.000,C 90.000,E1 7.587} C_DIS
LIN {X -0.042,Y -434.645,Z 732.829,A 0.000,B 0.000,C 90.000,E1 5.277} C_DIS
LIN {X -0.181,Y -438.482,Z 732.816,A 0.000,B 0.000,C 90.000,E1 2.980} C_DIS
LIN {X 0.187,Y -442.659,Z 732.804,A 0.000,B 0.000,C 90.000,E1 0.630} C_DIS
LIN {X -0.181,Y -446.814,Z 732.792,A 0.000,B 0.000,C 90.000,E1 358.511} C_DIS
LIN {X 0.181,Y -452.078,Z 732.777,A 0.000,B 0.000,C 90.000,E1 355.869} C_DIS
LIN {X -0.079,Y -456.310,Z 732.766,A 0.000,B 0.000,C 90.000,E1 353.970} C_DIS
LIN {X 0.025,Y -459.762,Z 732.758,A 0.000,B 0.000,C 90.000,E1 352.356} C_DIS
LIN {X -0.205,Y -463.162,Z 732.749,A 0.000,B 0.000,C 90.000,E1 350.792} C_DIS
LIN {X 0.163,Y -466.329,Z 732.740,A 0.000,B 0.000,C 90.000,E1 349.162} C_DIS
LIN {X 0.130,Y -469.340,Z 732.731,A 0.000,B 0.000,C 90.000,E1 347.589} C_DIS
LIN {X 0.181,Y -472.734,Z 732.721,A 0.000,B 0.000,C 90.000,E1 345.700} C_DIS
LIN {X -0.186,Y -476.810,Z 732.709,A 0.000,B 0.000,C 90.000,E1 343.559} C_DIS
LIN {X -0.118,Y -479.424,Z 732.702,A 0.000,B 0.000,C 90.000,E1 342.308} C_DIS
LIN {X 0.142,Y -481.955,Z 732.697,A 0.000,B 0.000,C 90.000,E1 341.348} C_DIS
LIN {X 0.135,Y -482.954,Z 732.695,A 0.000,B 0.000,C 90.000,E1 341.040} C_DIS
LIN {X 0.137,Y -485.772,Z 732.691,A 0.000,B 0.000,C 90.000,E1 340.423} C_DIS
LIN {X -0.118,Y -488.112,Z 732.689,A 0.000,B 0.000,C 90.000,E1 340.061} C_DIS
LIN {X -0.099,Y -490.346,Z 732.688,A 0.000,B 0.000,C 90.000,E1 339.752} C_DIS
END
